# B&R Automation Studio project EFI
Automation Studio 4.12.6.106; Program for EFI Printing Machines; technology packages: Acp10Arnc0 5.21.2, mapp 5.21.0, mappView 5.21.0

## Configuration 1BK2Bar

CPU X20CP1382, AutomationRuntime B4.83, Build 4.1.2, Safety 1.10

### Task classes (Cpu.sw)
```
Cyclic#1 (cycle 4000 us, tolerance 0 us):
  InitSteprs <- ExtPack._Motion.StepperCtrl.StepperCtrl_v1.InitStepperX2XCtrl.prg (BuildOptions=-D _IGNORE_CHECKLIB)
  Stepper3L1 <- ExtPack._Motion.StepperCtrl.StepperCtrl_v1.StepperX2XCtrl.prg (BuildOptions=-D _IGNORE_CHECKLIB)
  Stepper3L2 <- ExtPack._Motion.StepperCtrl.StepperCtrl_v1.StepperX2XCtrl.prg (BuildOptions=-D _IGNORE_CHECKLIB)
  Analog <- (binary) (BuildOptions=-D _IGNORE_CHECKLIB)
  Visu_Inks <- (binary) (BuildOptions=-D _IGNORE_CHECKLIB)
  Slave_mbus <- (binary) (BuildOptions=-D _IGNORE_CHECKLIB)
Cyclic#2 (cycle 12000 us, tolerance 0 us):
  Initialize <- Printer.Config.Initialize.prg (BuildOptions=-D _IGNORE_CHECKLIB)
  InitAxis <- ExtPack._Motion.AxisCtrl.AxisCtrl_v2.InitAxisControl.prg (BuildOptions=-D _IGNORE_CHECKLIB)
  Belt <- ExtPack._Motion.AxisCtrl.AxisCtrl_v2.AxisCtrl.prg (BuildOptions=-D _IGNORE_CHECKLIB)
  BK_A <- ExtPack._Motion.AxisCtrl.AxisCtrl_v2.AxisCtrl.prg (BuildOptions=-D _IGNORE_CHECKLIB)
  Stepper3L <- ExtPack._Motion.AxisCtrl.AxisCtrl_v2.AxisCtrl.prg (BuildOptions=-D _IGNORE_CHECKLIB)
  Gear3L <- ExtPack._Motion.AxisCtrl.AxisCtrl_v2.AxisCtrl.prg (BuildOptions=-D _IGNORE_CHECKLIB)
  InitIcla <- ExtPack._Motion.IclaCtrl.IclaCtrl_v4.InitIclaCtrl.prg (BuildOptions=-D _IGNORE_CHECKLIB)
  IclaBK_A <- ExtPack._Motion.IclaCtrl.IclaCtrl_v4.IclaCtrl.prg (BuildOptions=-D _IGNORE_CHECKLIB)
  Analog_Fas <- ExtPack._Media.AnalogThicknessCtrl.AnalogThicknessCtrl_v1.Analog_Fast.prg (BuildOptions=-D _IGNORE_CHECKLIB)
  nSens_Fast <- ExtPack._Media.nSensorCtrl.nSensorCtrl_v2.nSensorCtrl_Fast.prg (BuildOptions=-D _IGNORE_CHECKLIB)
  Thick_Fast <- ExtPack._Media.ThicknessCtrl.ThicknessCtrl_v2.ThicknessCtrl_Fast.prg (BuildOptions=-D _IGNORE_CHECKLIB)
Cyclic#4 (cycle 32000 us, tolerance 32000 us):
  PhysInput <- Printer.PhysicalMapping.PhysicalMapInputs.prg (BuildOptions=-D _IGNORE_CHECKLIB)
  BlockInp <- Printer.BlockSignalsManager.BlockInputsMapping.prg (BuildOptions=-D _IGNORE_CHECKLIB)  // Physical inputs/outputs block
  ThickPos <- ExtPack._Media.ThicknessCtrl.ThicknessCtrl_v2.ThicknessCtrl.prg (BuildOptions=-D _IGNORE_CHECKLIB)  // Thickness array manager
  Mach_Fast <- Printer.MachineCtrl.MachineCtrl_Fast.prg (BuildOptions=-D _IGNORE_CHECKLIB)
  BeltCtrl <- ExtPack._Transport.BeltCtrl.BeltCtrl_v1.BeltCtrl.prg (BuildOptions=-D _IGNORE_CHECKLIB)  // Belt program
  InitBlockC <- ExtPack.BlockCtrl.BlockCtrl_v1.InitBlockCtrl.prg (BuildOptions=-D _IGNORE_CHECKLIB)  // Init blocks
  Block_BK1 <- ExtPack.BlockCtrl.BlockCtrl_v1.BlockCtrl.prg (BuildOptions=-D _IGNORE_CHECKLIB)
  AnalogThic <- ExtPack._Media.AnalogThicknessCtrl.AnalogThicknessCtrl_v1.AnalogThickness.prg (BuildOptions=-D _IGNORE_CHECKLIB)
  nSensorCtr <- ExtPack._Media.nSensorCtrl.nSensorCtrl_v2.nSensorCtrl.prg (BuildOptions=-D _IGNORE_CHECKLIB)
  InitChille <- ExtPack._Extras.ChillerCtrl.ChillerCtrl_v2.InitChiller.prg (BuildOptions=-D _IGNORE_CHECKLIB)
  ChillCtr1 <- ExtPack._Extras.ChillerCtrl.ChillerCtrl_v2.ChillerCtrl.prg (BuildOptions=-D _IGNORE_CHECKLIB)
  BlockOut <- Printer.BlockSignalsManager.BlockOutputsMapping.prg (BuildOptions=-D _IGNORE_CHECKLIB)  // Physical HW outputs
  PhysOutput <- Printer.PhysicalMapping.PhysicalMapOutputs.prg (BuildOptions=-D _IGNORE_CHECKLIB)
Cyclic#5 (cycle 80000 us, tolerance 80000 us):
  InksInputs <- Printer.InksSignals.InksInputs.prg (BuildOptions=-D _IGNORE_CHECKLIB)  // Physical inputs inks
  InitIndex <- ExtPack.InksCtrl.InksCtrl_v3.InitInksCtrl.prg (BuildOptions=-D _IGNORE_CHECKLIB)
  Inks_01 <- ExtPack.InksCtrl.InksCtrl_v3.InksCtrl.prg (BuildOptions=-D _IGNORE_CHECKLIB)
  Inks_02 <- ExtPack.InksCtrl.InksCtrl_v3.InksCtrl.prg (BuildOptions=-D _IGNORE_CHECKLIB)
  InksOutput <- Printer.InksSignals.InksOutputs.prg (BuildOptions=-D _IGNORE_CHECKLIB)  // Physical outputs inks
  SafetySamp <- AsSafetySolution.SafetySample.prg (BuildOptions=-D _IGNORE_CHECKLIB)
  EventLogGe <- ExtPack._Tools.EventLog.EventLog_v1.EventLogGen.prg (BuildOptions=-D _IGNORE_CHECKLIB)
  SavePerman <- Printer.Config.SavePermanent.prg (BuildOptions=-D _IGNORE_CHECKLIB)
Cyclic#6 (cycle 88000 us, tolerance 88000 us):
  Mach_Conf <- Printer.Config.MachineConfigurator.prg (BuildOptions=-D _IGNORE_CHECKLIB)  // Printer configurator program
  Mach_Slow <- Printer.MachineCtrl.MachineCtrl_Slow.prg (BuildOptions=-D _IGNORE_CHECKLIB)
Cyclic#7 (cycle 44000 us, tolerance 88000 us):
  PLC2Kernel <- Printer.Comms.PLC2Kernel.prg (BuildOptions=-D _IGNORE_CHECKLIB)  // Comn PLC to kernel
  ServModbus <- ExtPack._Comms.ModbusComms.ModbusComms_v1.ServModbus.prg (BuildOptions=-D _IGNORE_CHECKLIB)
  Kernel2PLC <- Printer.Comms.Kernel2PLC.prg (BuildOptions=-D _IGNORE_CHECKLIB)  // Comns Kernel to PLC
Cyclic#8 (cycle 200000 us):
  NwSNTPClie <- ExtPack._Comms.SNTPClient.SNTPClient_v1.NwSNTPClient.prg [disabled] (BuildOptions=-D _IGNORE_CHECKLIB)
DataObjects: Acp10sys, assl1
NcDataObjects: AcpErrTxt <- AxisTables.AcpErrTxt.dob, acp10etxen <- AxisTables.acp10etxen.dob, BeltP4_a <- AxisTables.BeltP4_a.dob, BeltP4_i <- AxisTables.BeltP4_i.dob, BeltShield <- AxisTables.BeltShield_a.dob, BeltShiel1 <- AxisTables.BeltShield_i.dob, BK1_a <- AxisTables.BK1_a.dob, BK1_i <- AxisTables.BK1_i.dob, SM_a <- AxisTables.SM_a.dob, SM_i <- AxisTables.SM_i.dob
Binaries: udbdef, TCData, mvLoader, TCLang, Acp10map, acp10cfg, iomap, User, ashwac, arconfig, Role, ashwd, sysconf, asfw, vccnum, vcpdvnc, Visu02, vccalarm, vccovl, vcshared, vcfile, Panel101, vccstr, vccline, arial, vcpfx20, vcchtml, vcgclass, vccbtn, vcrt, Visu03, vcctext, vcclbox, Panel102, vccbmp, vcfntttf, vcctrend, vcalarm, vcdsint, vcnet, vccshape, arialbd, vctcal, Panel103, vcmgr, vcdsloc, Visu01, vcpkat, vccurl, vccdt, vccbar, vcpdsw, vcxml, vcbclass, Diagn01, vccslider, vccddbox, Diagn02, vccpopup, vcchspot, Diagn03
Libraries: AsCANopen, FBs, Functions, ConvertFun, runtime, brsystem, sys_lib, standard, AsSafety, FileIO, AsXml, astime, asstring, AsFifo, NcGlobal, AsBrStr, MTBasics, MTTypes, MTFilter, AsTCP, AsIecCon, AsIOAcc, AsBrMath, AsEPL, ArEventLog, Acp10_MC, Acp10man, Acp10par, Acp10sim, Acp10sdc, DataObj, EvLogLib, BRSE_MB, BRSE_MBT, AxisFunc, AsSem, AsARCfg, ThickLib, powerlnk, arproject, arssl, asopcuas, asopcuac, vcresman, ashw
```

### Hardware
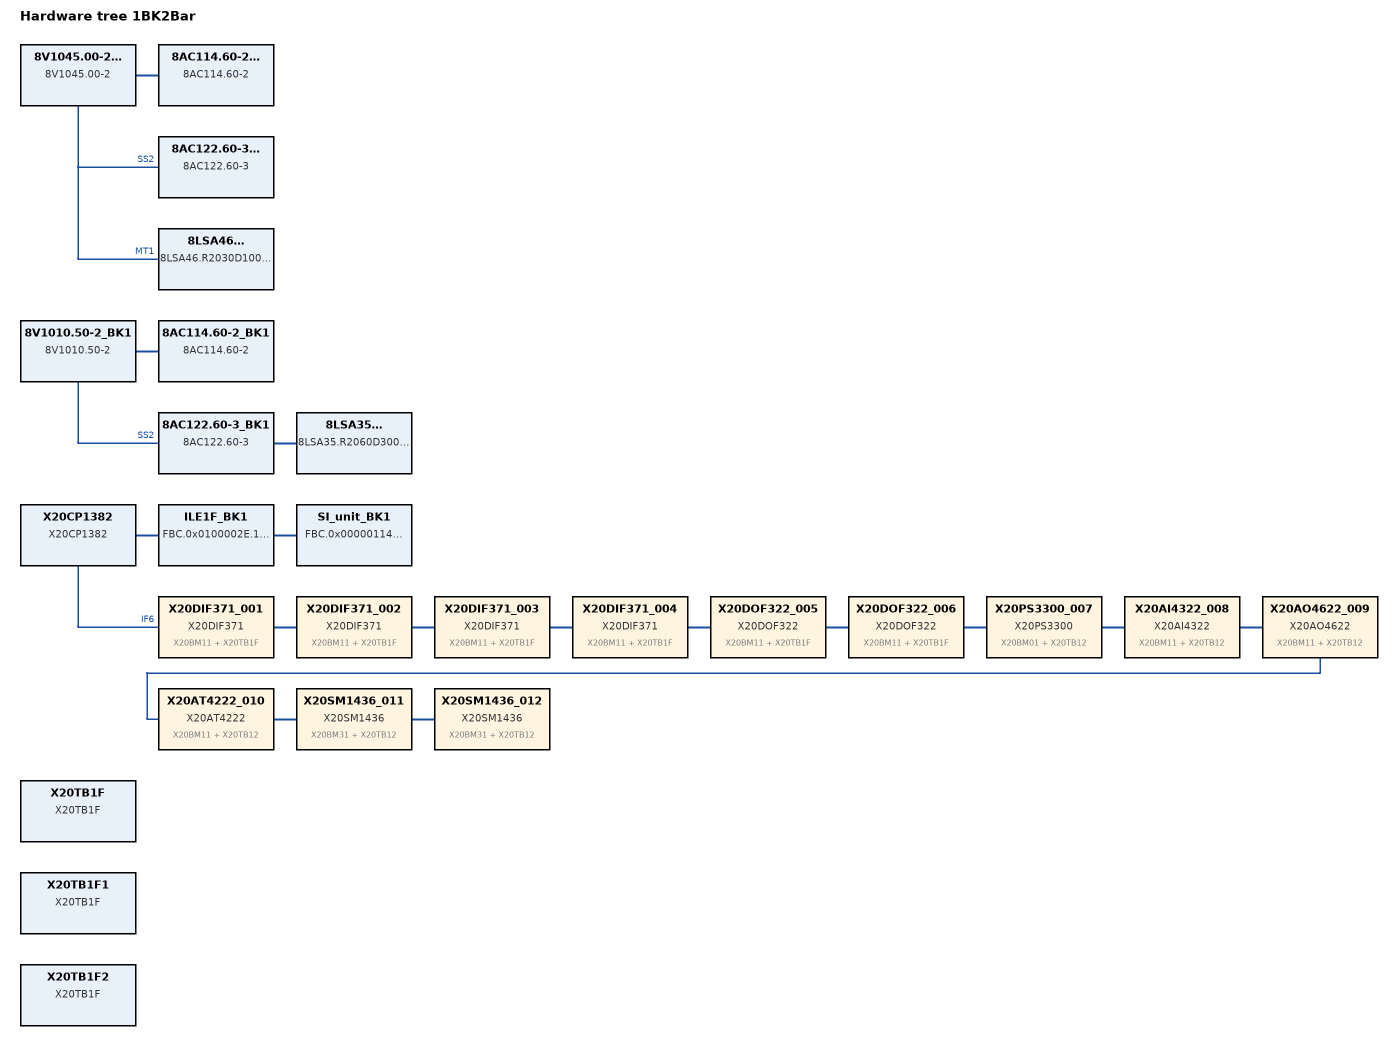
```
8AC114.60-2_BELT : 8AC114.60-2 v1.0.0.8  [SS -> 8V1045.00-2_BELT.SS1; PLK1 -> 8AC114.60-2_BK1.PLK2 (NodeNumber=1) [Cable Type=PowerlinkCable, Length=10, Version=1.0.0.3]]
8AC114.60-2_BK1 : 8AC114.60-2 v1.0.0.8  [SS -> 8V1010.50-2_BK1.SS1; PLK1 -> X20CP1382.IF3 (NodeNumber=2) [Cable Type=PowerlinkCable, Length=10, Version=1.0.0.3]; PLK2 -> 8AC114.60-2_BELT.PLK1 (NodeNumber=2) [Cable Type=PowerlinkCable, Length=10, Version=1.0.0.3]]
8AC122.60-3_BELT : 8AC122.60-3 v2.2.0.0  [SS -> 8V1045.00-2_BELT.SS2]
8AC122.60-3_BK1 : 8AC122.60-3 v2.2.0.0  [SS -> 8V1010.50-2_BK1.SS2]
8LSA35.R2060D300-3 : 8LSA35.R2060D300-3 v1.0.4.39  [EC -> 8AC122.60-3_BK1.EC; MT -> 8V1010.50-2_BK1.MT1]
8LSA46.R2030D100-3 : 8LSA46.R2030D100-3 v2.2.0.0  [MT -> 8V1045.00-2_BELT.MT1]
8V1010.50-2_BK1 : 8V1010.50-2 v2.2.0.0
  SinglePhaseOperation = on
  BothEndSwitchesAreNormallyOpen_r1 = on
  QuickStopIsNormallyOpen_r1 = on
8V1045.00-2_BELT : 8V1045.00-2 v2.2.0.0
ILE1F_BK1 : FBC.0x0100002E.1.SEILE1F_0110E v1.10 (OrderNumber=ILE1F)  [CAN1 -> X20CP1382.IF7 (NodeNumber=5)]
  p1403_transmissionselection = 1
  plifeguarding_guardtime = 500
  plifeguarding_retryfactor = 10
  p3001_parametername = mandatory
  p3001_objecttype = 9
  p3001_subnumber = 0x3
  p3001_parametervalue = 
  p3001_objflags = 0
  p3001sub0_parametername = number of entries
  p3001sub0_objecttype = 7
  p3001sub0_datatype = 5
  p3001sub0_accesstype = ro
  p3001sub0_pdomapping = 0
  p3001sub1_parametername = Config.PrgNo
  p3001sub1_objecttype = 7
  p3001sub1_datatype = 7
  p3001sub1_lowlimit = 
  p3001sub1_highlimit = 
  p3001sub1_accesstype = ro
  p3001sub1_pdomapping = 0
  p3001sub2_parametername = Config.PrgVer
  p3001sub2_objecttype = 7
  p3001sub2_datatype = 7
  p3001sub2_lowlimit = 
  p3001sub2_highlimit = 
  p3001sub2_accesstype = ro
  p3001sub2_pdomapping = 0
  p300b_parametername = system settings
  p300b_objecttype = 9
  p300b_subnumber = 0x7
  p300b_parametervalue = 
  p300b_objflags = 0
  p300bsub0_parametername = number of entries
  p300bsub0_objecttype = 7
  p300bsub0_datatype = 5
  p300bsub0_accesstype = ro
  p300bsub0_pdomapping = 0
  p300bsub1_parametername = Settings.name1
  p300bsub1_objecttype = 7
  p300bsub1_datatype = 7
  p300bsub1_lowlimit = 
  p300bsub1_highlimit = 
  p300bsub1_accesstype = rw
  p300bsub1_pdomapping = 0
  p300bsub1_parametervalue = 
  p300bsub1_objflags = 0
  p300bsub2_parametername = Settings.name2
  p300bsub2_objecttype = 7
  p300bsub2_datatype = 7
  p300bsub2_lowlimit = 
  p300bsub2_highlimit = 
  p300bsub2_accesstype = rw
  p300bsub2_pdomapping = 0
  p300bsub2_parametervalue = 
  p300bsub2_objflags = 0
  p300bsub6_parametername = Commands.eeprSave
  p300bsub6_objecttype = 7
  p300bsub6_datatype = 6
  p300bsub6_lowlimit = 
  p300bsub6_highlimit = 
  p300bsub6_accesstype = rw
  p300bsub6_pdomapping = 0
  p300bsub6_parametervalue = 1
  p300bsub6_objflags = 0
  p300bsub7_parametername = Commands.stateSave
  p300bsub7_objecttype = 7
  p300bsub7_datatype = 6
  p300bsub7_lowlimit = 
  p300bsub7_highlimit = 
  p300bsub7_accesstype = ro
  p300bsub7_pdomapping = 0
  p300bsub8_parametername = Commands.default
  p300bsub8_objecttype = 7
  p300bsub8_datatype = 6
  p300bsub8_lowlimit = 
  p300bsub8_highlimit = 
  p300bsub8_accesstype = rw
  p300bsub8_pdomapping = 0
  p300bsub8_parametervalue = 
  p300bsub8_objflags = 0
  p300bsub9_parametername = Commands.stateDef
  p300bsub9_objecttype = 7
  p300bsub9_datatype = 6
  p300bsub9_lowlimit = 
  p300bsub9_highlimit = 
  p300bsub9_accesstype = ro
  p300bsub9_pdomapping = 0
  p300f_parametername = controller  settings
  p300f_objecttype = 9
  p300f_subnumber = 0xE
  p300f_parametervalue = 
  p300f_objflags = 0
  p300fsub0_parametername = number of entries
  p300fsub0_objecttype = 7
  p300fsub0_datatype = 5
  p300fsub0_accesstype = ro
  p300fsub0_pdomapping = 0
  p300fsub1_parametername = Config.I_nomDrv
  p300fsub1_objecttype = 7
  p300fsub1_datatype = 6
  p300fsub1_accesstype = ro
  p300fsub1_pdomapping = 0
  p300fsub2_parametername = Config.I_maxDrv
  p300fsub2_objecttype = 7
  p300fsub2_datatype = 6
  p300fsub2_accesstype = ro
  p300fsub2_pdomapping = 0
  p300fsub3_parametername = Settings.I_max
  p300fsub3_objecttype = 7
  p300fsub3_datatype = 6
  p300fsub3_accesstype = rw
  p300fsub3_pdomapping = 0
  p300fsub3_parametervalue = 60
  p300fsub3_objflags = 0
  p300fsub5_parametername = Settings.I_maxBlk
  p300fsub5_objecttype = 7
  p300fsub5_datatype = 6
  p300fsub5_lowlimit = 
  p300fsub5_highlimit = 
  p300fsub5_accesstype = rw
  p300fsub5_pdomapping = 0
  p300fsub5_parametervalue = 20
  p300fsub5_objflags = 0
  p300fsub7_parametername = Settings.p_maxDiff
  p300fsub7_objecttype = 7
  p300fsub7_datatype = 6
  p300fsub7_lowlimit = 
  p300fsub7_highlimit = 
  p300fsub7_accesstype = rw
  p300fsub7_pdomapping = 0
  p300fsub7_parametervalue = 24
  p300fsub7_objflags = 0
  p300fsub8_parametername = Control.KPn
  p300fsub8_objecttype = 7
  p300fsub8_datatype = 6
  p300fsub8_lowlimit = 
  p300fsub8_highlimit = 
  p300fsub8_accesstype = rw
  p300fsub8_pdomapping = 0
  p300fsub8_parametervalue = 60
  p300fsub8_objflags = 0
  p300fsub9_parametername = Control.TNn
  p300fsub9_objecttype = 7
  p300fsub9_datatype = 6
  p300fsub9_lowlimit = 
  p300fsub9_highlimit = 
  p300fsub9_accesstype = rw
  p300fsub9_pdomapping = 0
  p300fsub9_parametervalue = 10000
  p300fsub9_objflags = 0
  p300fsuba_parametername = Control.KPp
  p300fsuba_objecttype = 7
  p300fsuba_datatype = 6
  p300fsuba_lowlimit = 
  p300fsuba_highlimit = 
  p300fsuba_accesstype = rw
  p300fsuba_pdomapping = 0
  p300fsuba_parametervalue = 300
  p300fsuba_objflags = 0
  p300fsubb_parametername = Control.KFPp
  p300fsubb_objecttype = 7
  p300fsubb_datatype = 6
  p300fsubb_lowlimit = 
  p300fsubb_highlimit = 
  p300fsubb_accesstype = rw
  p300fsubb_pdomapping = 0
  p300fsubb_parametervalue = 32767
  p300fsubb_objflags = 0
  p300fsubc_parametername = Settings.T_block
  p300fsubc_objecttype = 7
  p300fsubc_datatype = 6
  p300fsubc_lowlimit = 
  p300fsubc_highlimit = 
  p300fsubc_accesstype = rw
  p300fsubc_pdomapping = 0
  p300fsubc_parametervalue = 100
  p300fsubc_objflags = 0
  p300fsubd_parametername = Status.p_difPeak
  p300fsubd_objecttype = 7
  p300fsubd_datatype = 7
  p300fsubd_lowlimit = 
  p300fsubd_highlimit = 
  p300fsubd_accesstype = rw
  p300fsubd_pdomapping = 0
  p300fsubd_parametervalue = 
  p300fsubd_objflags = 0
  p300fsubf_parametername = Settings.p_win
  p300fsubf_objecttype = 7
  p300fsubf_datatype = 6
  p300fsubf_lowlimit = 
  p300fsubf_highlimit = 
  p300fsubf_accesstype = rw
  p300fsubf_pdomapping = 0
  p300fsubf_parametervalue = 1
  p300fsubf_objflags = 0
  p300fsub10_parametername = Settings.p_winTime
  p300fsub10_objecttype = 7
  p300fsub10_datatype = 6
  p300fsub10_lowlimit = 
  p300fsub10_highlimit = 
  p300fsub10_accesstype = rw
  p300fsub10_pdomapping = 0
  p300fsub10_parametervalue = 0
  p300fsub10_objflags = 0
  p3016_parametername = rs485
  p3016_objecttype = 9
  p3016_subnumber = 0x4
  p3016_parametervalue = 
  p3016_objflags = 0
  p3016sub0_parametername = number of entries
  p3016sub0_objecttype = 7
  p3016sub0_datatype = 5
  p3016sub0_accesstype = ro
  p3016sub0_pdomapping = 0
  p3016sub1_parametername = RS485.serBaud
  p3016sub1_objecttype = 7
  p3016sub1_datatype = 6
  p3016sub1_lowlimit = 
  p3016sub1_highlimit = 
  p3016sub1_accesstype = rw
  p3016sub1_pdomapping = 0
  p3016sub1_parametervalue = 
  p3016sub1_objflags = 0
  p3016sub2_parametername = RS485.serAdr
  p3016sub2_objecttype = 7
  p3016sub2_datatype = 6
  p3016sub2_lowlimit = 
  p3016sub2_highlimit = 
  p3016sub2_accesstype = rw
  p3016sub2_pdomapping = 0
  p3016sub2_parametervalue = 
  p3016sub2_objflags = 0
  p3016sub3_parametername = RS485.serFormat
  p3016sub3_objecttype = 7
  p3016sub3_datatype = 6
  p3016sub3_lowlimit = 
  p3016sub3_highlimit = 
  p3016sub3_accesstype = rw
  p3016sub3_pdomapping = 0
  p3016sub3_parametervalue = 
  p3016sub3_objflags = 0
  p3017_parametername = can
  p3017_objecttype = 9
  p3017_subnumber = 0x3
  p3017_parametervalue = 
  p3017_objflags = 0
  p3017sub0_parametername = number of entries
  p3017sub0_objecttype = 7
  p3017sub0_datatype = 5
  p3017sub0_accesstype = ro
  p3017sub0_pdomapping = 0
  p3017sub2_parametername = CAN.canAddr
  p3017sub2_objecttype = 7
  p3017sub2_datatype = 6
  p3017sub2_lowlimit = 
  p3017sub2_highlimit = 
  p3017sub2_accesstype = rw
  p3017sub2_pdomapping = 0
  p3017sub2_parametervalue = 
  p3017sub2_objflags = 0
  p3017sub3_parametername = CAN.canBaud
  p3017sub3_objecttype = 7
  p3017sub3_datatype = 6
  p3017sub3_lowlimit = 
  p3017sub3_highlimit = 
  p3017sub3_accesstype = rw
  p3017sub3_pdomapping = 0
  p3017sub3_parametervalue = 
  p3017sub3_objflags = 0
  p301c_parametername = settings1
  p301c_objecttype = 9
  p301c_subnumber = 0xF
  p301c_parametervalue = 
  p301c_objflags = 0
  p301csub0_parametername = number of entries
  p301csub0_objecttype = 7
  p301csub0_datatype = 5
  p301csub0_accesstype = ro
  p301csub0_pdomapping = 0
  p301csub3_parametername = Status.xMode_act
  p301csub3_objecttype = 7
  p301csub3_datatype = 6
  p301csub3_lowlimit = 
  p301csub3_highlimit = 
  p301csub3_accesstype = ro
  p301csub3_pdomapping = 0
  p301csub6_parametername = Motion.invertDir
  p301csub6_objecttype = 7
  p301csub6_datatype = 6
  p301csub6_lowlimit = 
  p301csub6_highlimit = 
  p301csub6_accesstype = rw
  p301csub6_pdomapping = 0
  p301csub6_parametervalue = 0
  p301csub6_objflags = 0
  p301csuba_parametername = Status.WarnSig
  p301csuba_objecttype = 7
  p301csuba_datatype = 6
  p301csuba_lowlimit = 
  p301csuba_highlimit = 
  p301csuba_accesstype = ro
  p301csuba_pdomapping = 0
  p301csubb_parametername = Settings.WarnOvrun
  p301csubb_objecttype = 7
  p301csubb_datatype = 6
  p301csubb_lowlimit = 
  p301csubb_highlimit = 
  p301csubb_accesstype = rw
  p301csubb_pdomapping = 0
  p301csubb_parametervalue = 0
  p301csubb_objflags = 0
  p301csubd_parametername = Settings.SignEnabl
  p301csubd_objecttype = 7
  p301csubd_datatype = 6
  p301csubd_lowlimit = 
  p301csubd_highlimit = 
  p301csubd_accesstype = rw
  p301csubd_pdomapping = 0
  p301csubd_parametervalue = 3
  p301csubd_objflags = 0
  p301csube_parametername = Settings.SignLevel
  p301csube_objecttype = 7
  p301csube_datatype = 6
  p301csube_lowlimit = 
  p301csube_highlimit = 
  p301csube_accesstype = rw
  p301csube_pdomapping = 0
  p301csube_parametervalue = 0
  p301csube_objflags = 0
  p301csubf_parametername = Status.Sign_SR
  p301csubf_objecttype = 7
  p301csubf_datatype = 6
  p301csubf_lowlimit = 
  p301csubf_highlimit = 
  p301csubf_accesstype = ro
  p301csubf_pdomapping = 0
  p301csub11_parametername = Status.FltSig
  p301csub11_objecttype = 7
  p301csub11_datatype = 7
  p301csub11_lowlimit = 
  p301csub11_highlimit = 
  p301csub11_accesstype = ro
  p301csub11_pdomapping = 0
  p301csub12_parametername = Status.FltSig_SR
  p301csub12_objecttype = 7
  p301csub12_datatype = 7
  p301csub12_lowlimit = 
  p301csub12_highlimit = 
  p301csub12_accesstype = ro
  p301csub12_pdomapping = 0
  p301csub13_parametername = Status.action_st
  p301csub13_objecttype = 7
  p301csub13_datatype = 6
  p301csub13_lowlimit = 
  p301csub13_highlimit = 
  p301csub13_accesstype = ro
  p301csub13_pdomapping = 0
  p301csub15_parametername = Motion.dec_Stop
  p301csub15_objecttype = 7
  p301csub15_datatype = 7
  p301csub15_lowlimit = 
  p301csub15_highlimit = 
  p301csub15_accesstype = rw
  p301csub15_pdomapping = 0
  p301csub15_parametervalue = 4960
  p301csub15_objflags = 0
  p301csub18_parametername = Settings.Flt_pDiff
  p301csub18_objecttype = 7
  p301csub18_datatype = 6
  p301csub18_lowlimit = 
  p301csub18_highlimit = 
  p301csub18_accesstype = rw
  p301csub18_pdomapping = 0
  p301csub18_parametervalue = 3
  p301csub18_objflags = 0
  p301d_parametername = settings2
  p301d_objecttype = 9
  p301d_subnumber = 0x4
  p301d_parametervalue = 
  p301d_objflags = 0
  p301dsub0_parametername = number of entries
  p301dsub0_objecttype = 7
  p301dsub0_datatype = 5
  p301dsub0_accesstype = ro
  p301dsub0_pdomapping = 0
  p301dsub2_parametername = Config.ResolutM
  p301dsub2_objecttype = 7
  p301dsub2_datatype = 6
  p301dsub2_accesstype = ro
  p301dsub2_pdomapping = 0
  p301dsub17_parametername = Motion.v_target0
  p301dsub17_objecttype = 7
  p301dsub17_datatype = 6
  p301dsub17_accesstype = rw
  p301dsub17_pdomapping = 0
  p301dsub17_parametervalue = 1000
  p301dsub17_objflags = 0
  p301dsub1a_parametername = Motion.acc
  p301dsub1a_objecttype = 7
  p301dsub1a_datatype = 7
  p301dsub1a_lowlimit = 
  p301dsub1a_highlimit = 
  p301dsub1a_accesstype = rw
  p301dsub1a_pdomapping = 0
  p301dsub1a_parametervalue = 2442
  p301dsub1a_objflags = 0
  p301e_parametername = pdo data
  p301e_objecttype = 9
  p301e_subnumber = 0xC
  p301e_parametervalue = 
  p301e_objflags = 0
  p301esub0_parametername = number of entries
  p301esub0_objecttype = 7
  p301esub0_datatype = 5
  p301esub0_accesstype = ro
  p301esub0_pdomapping = 0
  p301esubb_parametername = Status.ModeError
  p301esubb_objecttype = 7
  p301esubb_datatype = 6
  p301esubb_lowlimit = 
  p301esubb_highlimit = 
  p301esubb_accesstype = ro
  p301esubb_pdomapping = 0
  p301f_parametername = status
  p301f_objecttype = 9
  p301f_subnumber = 0x11
  p301f_parametervalue = 
  p301f_objflags = 0
  p301fsub0_parametername = number of entries
  p301fsub0_objecttype = 7
  p301fsub0_datatype = 5
  p301fsub0_accesstype = ro
  p301fsub0_pdomapping = 0
  p301fsub1_parametername = Status.v_ref
  p301fsub1_objecttype = 7
  p301fsub1_datatype = 4
  p301fsub1_lowlimit = 
  p301fsub1_highlimit = 
  p301fsub1_accesstype = ro
  p301fsub1_pdomapping = 0
  p301fsub2_parametername = Status.v_act
  p301fsub2_objecttype = 7
  p301fsub2_datatype = 4
  p301fsub2_lowlimit = 
  p301fsub2_highlimit = 
  p301fsub2_accesstype = ro
  p301fsub2_pdomapping = 0
  p301fsub5_parametername = Status.p_ref
  p301fsub5_objecttype = 7
  p301fsub5_datatype = 4
  p301fsub5_lowlimit = 
  p301fsub5_highlimit = 
  p301fsub5_accesstype = ro
  p301fsub5_pdomapping = 0
  p301fsub6_parametername = Status.p_act
  p301fsub6_objecttype = 7
  p301fsub6_datatype = 4
  p301fsub6_lowlimit = 
  p301fsub6_highlimit = 
  p301fsub6_accesstype = ro
  p301fsub6_pdomapping = 0
  p301fsub7_parametername = Status.p_dif
  p301fsub7_objecttype = 7
  p301fsub7_datatype = 4
  p301fsub7_lowlimit = 
  p301fsub7_highlimit = 
  p301fsub7_accesstype = ro
  p301fsub7_pdomapping = 0
  p301fsub8_parametername = Status.n_ref
  p301fsub8_objecttype = 7
  p301fsub8_datatype = 3
  p301fsub8_lowlimit = 
  p301fsub8_highlimit = 
  p301fsub8_accesstype = ro
  p301fsub8_pdomapping = 0
  p301fsub9_parametername = Status.n_act
  p301fsub9_objecttype = 7
  p301fsub9_datatype = 3
  p301fsub9_lowlimit = 
  p301fsub9_highlimit = 
  p301fsub9_accesstype = ro
  p301fsub9_pdomapping = 0
  p301fsubc_parametername = Status.I_act
  p301fsubc_objecttype = 7
  p301fsubc_datatype = 3
  p301fsubc_lowlimit = 
  p301fsubc_highlimit = 
  p301fsubc_accesstype = ro
  p301fsubc_pdomapping = 0
  p301fsub14_parametername = Status.UDC_act
  p301fsub14_objecttype = 7
  p301fsub14_datatype = 6
  p301fsub14_lowlimit = 
  p301fsub14_highlimit = 
  p301fsub14_accesstype = ro
  p301fsub14_pdomapping = 0
  p301fsub19_parametername = Status.TPA_act
  p301fsub19_objecttype = 7
  p301fsub19_datatype = 6
  p301fsub19_lowlimit = 
  p301fsub19_highlimit = 
  p301fsub19_accesstype = ro
  p301fsub19_pdomapping = 0
  p301fsub1c_parametername = Status.v_pref
  p301fsub1c_objecttype = 7
  p301fsub1c_datatype = 4
  p301fsub1c_lowlimit = 
  p301fsub1c_highlimit = 
  p301fsub1c_accesstype = ro
  p301fsub1c_pdomapping = 0
  p301fsub1e_parametername = Status.p_target
  p301fsub1e_objecttype = 7
  p301fsub1e_datatype = 4
  p301fsub1e_lowlimit = 
  p301fsub1e_highlimit = 
  p301fsub1e_accesstype = ro
  p301fsub1e_pdomapping = 0
  p301fsub1f_parametername = Status.p_profile
  p301fsub1f_objecttype = 7
  p301fsub1f_datatype = 4
  p301fsub1f_lowlimit = 
  p301fsub1f_highlimit = 
  p301fsub1f_accesstype = ro
  p301fsub1f_pdomapping = 0
  p301fsub23_parametername = Status.n_profile
  p301fsub23_objecttype = 7
  p301fsub23_datatype = 3
  p301fsub23_lowlimit = 
  p301fsub23_highlimit = 
  p301fsub23_accesstype = ro
  p301fsub23_pdomapping = 0
  p301fsub26_parametername = Status.n_target
  p301fsub26_objecttype = 7
  p301fsub26_datatype = 3
  p301fsub26_lowlimit = 
  p301fsub26_highlimit = 
  p301fsub26_accesstype = ro
  p301fsub26_pdomapping = 0
  p301fsub2d_parametername = Status.n_pref
  p301fsub2d_objecttype = 7
  p301fsub2d_datatype = 3
  p301fsub2d_lowlimit = 
  p301fsub2d_highlimit = 
  p301fsub2d_accesstype = ro
  p301fsub2d_pdomapping = 0
  p3020_parametername = error
  p3020_objecttype = 9
  p3020_subnumber = 0x5
  p3020_parametervalue = 
  p3020_objflags = 0
  p3020sub0_parametername = number of entries
  p3020sub0_objecttype = 7
  p3020sub0_datatype = 5
  p3020sub0_accesstype = ro
  p3020sub0_pdomapping = 0
  p3020sub1_parametername = ErrorMemAvailable
  p3020sub1_objecttype = 7
  p3020sub1_datatype = 6
  p3020sub1_lowlimit = 
  p3020sub1_highlimit = 
  p3020sub1_accesstype = ro
  p3020sub1_pdomapping = 0
  p3020sub2_parametername = Commands.del_err
  p3020sub2_objecttype = 7
  p3020sub2_datatype = 6
  p3020sub2_lowlimit = 
  p3020sub2_highlimit = 
  p3020sub2_accesstype = rw
  p3020sub2_pdomapping = 0
  p3020sub2_parametervalue = 
  p3020sub2_objflags = 0
  p3020sub6_parametername = PowerOnCount
  p3020sub6_objecttype = 7
  p3020sub6_datatype = 7
  p3020sub6_lowlimit = 
  p3020sub6_highlimit = 
  p3020sub6_accesstype = ro
  p3020sub6_pdomapping = 0
  p3020sub7_parametername = Status.StopFault
  p3020sub7_objecttype = 7
  p3020sub7_datatype = 6
  p3020sub7_lowlimit = 
  p3020sub7_highlimit = 
  p3020sub7_accesstype = ro
  p3020sub7_pdomapping = 0
  p3021_parametername = io
  p3021_objecttype = 9
  p3021_subnumber = 0x4
  p3021_parametervalue = 
  p3021_objflags = 0
  p3021sub0_parametername = number of entries
  p3021sub0_objecttype = 7
  p3021sub0_datatype = 5
  p3021sub0_accesstype = ro
  p3021sub0_pdomapping = 0
  p3021sub1_parametername = I/O.IO_act
  p3021sub1_objecttype = 7
  p3021sub1_datatype = 6
  p3021sub1_lowlimit = 
  p3021sub1_highlimit = 
  p3021sub1_accesstype = rw
  p3021sub1_pdomapping = 0
  p3021sub1_parametervalue = 
  p3021sub1_objflags = 0
  p3021sub7_parametername = Commands.brake
  p3021sub7_objecttype = 7
  p3021sub7_datatype = 6
  p3021sub7_lowlimit = 
  p3021sub7_highlimit = 
  p3021sub7_accesstype = rw
  p3021sub7_pdomapping = 0
  p3021sub7_parametervalue = 
  p3021sub7_objflags = 0
  p3021sub8_parametername = Status.brake
  p3021sub8_objecttype = 7
  p3021sub8_datatype = 6
  p3021sub8_lowlimit = 
  p3021sub8_highlimit = 
  p3021sub8_accesstype = ro
  p3021sub8_pdomapping = 0
  p3022_parametername = io definitions
  p3022_objecttype = 9
  p3022_subnumber = 0x6
  p3022_parametervalue = 
  p3022_objflags = 0
  p3022sub0_parametername = number of entries
  p3022sub0_objecttype = 7
  p3022sub0_datatype = 5
  p3022sub0_accesstype = ro
  p3022sub0_pdomapping = 0
  p3022sub1_parametername = I/O.IO0_def
  p3022sub1_objecttype = 7
  p3022sub1_datatype = 6
  p3022sub1_lowlimit = 
  p3022sub1_highlimit = 
  p3022sub1_accesstype = rw
  p3022sub1_pdomapping = 0
  p3022sub1_parametervalue = 0
  p3022sub1_objflags = 0
  p3022sub2_parametername = I/O.IO1_def
  p3022sub2_objecttype = 7
  p3022sub2_datatype = 6
  p3022sub2_lowlimit = 
  p3022sub2_highlimit = 
  p3022sub2_accesstype = rw
  p3022sub2_pdomapping = 0
  p3022sub2_parametervalue = 0
  p3022sub2_objflags = 0
  p3022sub3_parametername = I/O.IO2_def
  p3022sub3_objecttype = 7
  p3022sub3_datatype = 6
  p3022sub3_lowlimit = 
  p3022sub3_highlimit = 
  p3022sub3_accesstype = rw
  p3022sub3_pdomapping = 0
  p3022sub3_parametervalue = 0
  p3022sub3_objflags = 0
  p3022sub4_parametername = I/O.IO3_def
  p3022sub4_objecttype = 7
  p3022sub4_datatype = 6
  p3022sub4_lowlimit = 
  p3022sub4_highlimit = 
  p3022sub4_accesstype = rw
  p3022sub4_pdomapping = 0
  p3022sub4_parametervalue = 
  p3022sub4_objflags = 0
  p3022sub7_parametername = I/O.progDelay
  p3022sub7_objecttype = 7
  p3022sub7_datatype = 6
  p3022sub7_lowlimit = 
  p3022sub7_highlimit = 
  p3022sub7_accesstype = rw
  p3022sub7_pdomapping = 0
  p3022sub7_parametervalue = 
  p3022sub7_objflags = 0
  p3023_parametername = ptp
  p3023_objecttype = 9
  p3023_subnumber = 0x6
  p3023_parametervalue = 
  p3023_objflags = 0
  p3023sub0_parametername = number of entries
  p3023sub0_objecttype = 7
  p3023sub0_datatype = 5
  p3023sub0_accesstype = ro
  p3023sub0_pdomapping = 0
  p3023sub1_parametername = PTP.p_absPTP
  p3023sub1_objecttype = 7
  p3023sub1_datatype = 4
  p3023sub1_lowlimit = 
  p3023sub1_highlimit = 
  p3023sub1_accesstype = rw
  p3023sub1_pdomapping = 0
  p3023sub1_parametervalue = 
  p3023sub1_objflags = 0
  p3023sub2_parametername = PTP.StatePTP
  p3023sub2_objecttype = 7
  p3023sub2_datatype = 6
  p3023sub2_lowlimit = 
  p3023sub2_highlimit = 
  p3023sub2_accesstype = ro
  p3023sub2_pdomapping = 0
  p3023sub3_parametername = PTP.p_relPTP
  p3023sub3_objecttype = 7
  p3023sub3_datatype = 4
  p3023sub3_lowlimit = 
  p3023sub3_highlimit = 
  p3023sub3_accesstype = rw
  p3023sub3_pdomapping = 0
  p3023sub3_parametervalue = 
  p3023sub3_objflags = 0
  p3023sub4_parametername = PTP.continue
  p3023sub4_objecttype = 7
  p3023sub4_datatype = 6
  p3023sub4_lowlimit = 
  p3023sub4_highlimit = 
  p3023sub4_accesstype = rw
  p3023sub4_pdomapping = 0
  p3023sub4_parametervalue = 
  p3023sub4_objflags = 0
  p3023sub5_parametername = PTP.v_tarPTP
  p3023sub5_objecttype = 7
  p3023sub5_datatype = 6
  p3023sub5_accesstype = rw
  p3023sub5_pdomapping = 0
  p3023sub5_parametervalue = 
  p3023sub5_objflags = 0
  p3024_parametername = vel
  p3024_objecttype = 9
  p3024_subnumber = 0x3
  p3024_parametervalue = 
  p3024_objflags = 0
  p3024sub0_parametername = number of entries
  p3024sub0_objecttype = 7
  p3024sub0_datatype = 5
  p3024sub0_accesstype = ro
  p3024sub0_pdomapping = 0
  p3024sub1_parametername = VEL.velocity
  p3024sub1_objecttype = 7
  p3024sub1_datatype = 3
  p3024sub1_accesstype = rw
  p3024sub1_pdomapping = 0
  p3024sub1_parametervalue = 
  p3024sub1_objflags = 0
  p3024sub2_parametername = VEL.stateVEL
  p3024sub2_objecttype = 7
  p3024sub2_datatype = 6
  p3024sub2_lowlimit = 
  p3024sub2_highlimit = 
  p3024sub2_accesstype = ro
  p3024sub2_pdomapping = 0
  p3028_parametername = homing
  p3028_objecttype = 9
  p3028_subnumber = 0xB
  p3028_parametervalue = 
  p3028_objflags = 0
  p3028sub0_parametername = number of entries
  p3028sub0_objecttype = 7
  p3028sub0_datatype = 5
  p3028sub0_accesstype = ro
  p3028sub0_pdomapping = 0
  p3028sub1_parametername = Homing.startHome
  p3028sub1_objecttype = 7
  p3028sub1_datatype = 6
  p3028sub1_lowlimit = 
  p3028sub1_highlimit = 
  p3028sub1_accesstype = rw
  p3028sub1_pdomapping = 0
  p3028sub1_parametervalue = 
  p3028sub1_objflags = 0
  p3028sub2_parametername = Homing.stateHome
  p3028sub2_objecttype = 7
  p3028sub2_datatype = 6
  p3028sub2_lowlimit = 
  p3028sub2_highlimit = 
  p3028sub2_accesstype = ro
  p3028sub2_pdomapping = 0
  p3028sub3_parametername = Homing.startSetp
  p3028sub3_objecttype = 7
  p3028sub3_datatype = 4
  p3028sub3_lowlimit = 
  p3028sub3_highlimit = 
  p3028sub3_accesstype = rw
  p3028sub3_pdomapping = 0
  p3028sub3_parametervalue = 
  p3028sub3_objflags = 0
  p3028sub4_parametername = Homing.v_Home
  p3028sub4_objecttype = 7
  p3028sub4_datatype = 6
  p3028sub4_accesstype = rw
  p3028sub4_pdomapping = 0
  p3028sub4_parametervalue = 
  p3028sub4_objflags = 0
  p3028sub5_parametername = Homing.v_outHome
  p3028sub5_objecttype = 7
  p3028sub5_datatype = 6
  p3028sub5_accesstype = rw
  p3028sub5_pdomapping = 0
  p3028sub5_parametervalue = 
  p3028sub5_objflags = 0
  p3028sub6_parametername = Homing.p_outHome
  p3028sub6_objecttype = 7
  p3028sub6_datatype = 4
  p3028sub6_lowlimit = 
  p3028sub6_highlimit = 
  p3028sub6_accesstype = rw
  p3028sub6_pdomapping = 0
  p3028sub6_parametervalue = 
  p3028sub6_objflags = 0
  p3028sub7_parametername = Homing.p_disHome
  p3028sub7_objecttype = 7
  p3028sub7_datatype = 4
  p3028sub7_lowlimit = 
  p3028sub7_highlimit = 
  p3028sub7_accesstype = rw
  p3028sub7_pdomapping = 0
  p3028sub7_parametervalue = 
  p3028sub7_objflags = 0
  p3028sub9_parametername = Homing.RefSwMod
  p3028sub9_objecttype = 7
  p3028sub9_datatype = 6
  p3028sub9_lowlimit = 
  p3028sub9_highlimit = 
  p3028sub9_accesstype = rw
  p3028sub9_pdomapping = 0
  p3028sub9_parametervalue = 
  p3028sub9_objflags = 0
  p3028subb_parametername = Homing.RefAppPos
  p3028subb_objecttype = 7
  p3028subb_datatype = 4
  p3028subb_lowlimit = 
  p3028subb_highlimit = 
  p3028subb_accesstype = rw
  p3028subb_pdomapping = 0
  p3028subb_parametervalue = 
  p3028subb_objflags = 0
  p3028subd_parametername = Homing.refError
  p3028subd_objecttype = 7
  p3028subd_datatype = 6
  p3028subd_lowlimit = 
  p3028subd_highlimit = 
  p3028subd_accesstype = ro
  p3028subd_pdomapping = 0
  p3029_parametername = manual
  p3029_objecttype = 9
  p3029_subnumber = 0x7
  p3029_parametervalue = 
  p3029_objflags = 0
  p3029sub0_parametername = number of entries
  p3029sub0_objecttype = 7
  p3029sub0_datatype = 5
  p3029sub0_accesstype = ro
  p3029sub0_pdomapping = 0
  p3029sub1_parametername = Manual.startMan
  p3029sub1_objecttype = 7
  p3029sub1_datatype = 6
  p3029sub1_lowlimit = 
  p3029sub1_highlimit = 
  p3029sub1_accesstype = rw
  p3029sub1_pdomapping = 0
  p3029sub1_parametervalue = 
  p3029sub1_objflags = 0
  p3029sub2_parametername = Manual.stateMan
  p3029sub2_objecttype = 7
  p3029sub2_datatype = 6
  p3029sub2_lowlimit = 
  p3029sub2_highlimit = 
  p3029sub2_accesstype = ro
  p3029sub2_pdomapping = 0
  p3029sub4_parametername = Manual.n_slowMan
  p3029sub4_objecttype = 7
  p3029sub4_datatype = 6
  p3029sub4_accesstype = rw
  p3029sub4_pdomapping = 0
  p3029sub4_parametervalue = 
  p3029sub4_objflags = 0
  p3029sub5_parametername = Manual.n_fastMan
  p3029sub5_objecttype = 7
  p3029sub5_datatype = 6
  p3029sub5_accesstype = rw
  p3029sub5_pdomapping = 0
  p3029sub5_parametervalue = 
  p3029sub5_objflags = 0
  p3029sub7_parametername = Manual.step_Man
  p3029sub7_objecttype = 7
  p3029sub7_datatype = 6
  p3029sub7_lowlimit = 
  p3029sub7_highlimit = 
  p3029sub7_accesstype = rw
  p3029sub7_pdomapping = 0
  p3029sub7_parametervalue = 
  p3029sub7_objflags = 0
  p3029sub8_parametername = Manual.time_Man
  p3029sub8_objecttype = 7
  p3029sub8_datatype = 6
  p3029sub8_lowlimit = 
  p3029sub8_highlimit = 
  p3029sub8_accesstype = rw
  p3029sub8_pdomapping = 0
  p3029sub8_parametervalue = 
  p3029sub8_objflags = 0
  p3320_parametername = prog io0
  p3320_objecttype = 9
  p3320_subnumber = 0x7
  p3320_parametervalue = 
  p3320_objflags = 0
  p3320sub0_parametername = number of entries
  p3320sub0_objecttype = 7
  p3320sub0_datatype = 5
  p3320sub0_accesstype = ro
  p3320sub0_pdomapping = 0
  p3320sub1_parametername = ProgIO0.Index
  p3320sub1_objecttype = 7
  p3320sub1_datatype = 6
  p3320sub1_lowlimit = 
  p3320sub1_highlimit = 
  p3320sub1_accesstype = rw
  p3320sub1_pdomapping = 0
  p3320sub1_parametervalue = 
  p3320sub1_objflags = 0
  p3320sub2_parametername = ProgIO0.Subindex
  p3320sub2_objecttype = 7
  p3320sub2_datatype = 6
  p3320sub2_lowlimit = 
  p3320sub2_highlimit = 
  p3320sub2_accesstype = rw
  p3320sub2_pdomapping = 0
  p3320sub2_parametervalue = 
  p3320sub2_objflags = 0
  p3320sub3_parametername = ProgIO0.BitMask
  p3320sub3_objecttype = 7
  p3320sub3_datatype = 7
  p3320sub3_lowlimit = 
  p3320sub3_highlimit = 
  p3320sub3_accesstype = rw
  p3320sub3_pdomapping = 0
  p3320sub3_parametervalue = 
  p3320sub3_objflags = 0
  p3320sub4_parametername = ProgIO0.Switch
  p3320sub4_objecttype = 7
  p3320sub4_datatype = 6
  p3320sub4_lowlimit = 
  p3320sub4_highlimit = 
  p3320sub4_accesstype = rw
  p3320sub4_pdomapping = 0
  p3320sub4_parametervalue = 
  p3320sub4_objflags = 0
  p3320sub5_parametername = ProgIO0.Value1
  p3320sub5_objecttype = 7
  p3320sub5_datatype = 4
  p3320sub5_lowlimit = 
  p3320sub5_highlimit = 
  p3320sub5_accesstype = rw
  p3320sub5_pdomapping = 0
  p3320sub5_parametervalue = 
  p3320sub5_objflags = 0
  p3320sub6_parametername = ProgIO0.Value2
  p3320sub6_objecttype = 7
  p3320sub6_datatype = 4
  p3320sub6_lowlimit = 
  p3320sub6_highlimit = 
  p3320sub6_accesstype = rw
  p3320sub6_pdomapping = 0
  p3320sub6_parametervalue = 
  p3320sub6_objflags = 0
  p3321_parametername = prog io1
  p3321_objecttype = 9
  p3321_subnumber = 0x7
  p3321_parametervalue = 
  p3321_objflags = 0
  p3321sub0_parametername = number of entries
  p3321sub0_objecttype = 7
  p3321sub0_datatype = 5
  p3321sub0_accesstype = ro
  p3321sub0_pdomapping = 0
  p3321sub1_parametername = ProgIO1.Index
  p3321sub1_objecttype = 7
  p3321sub1_datatype = 6
  p3321sub1_lowlimit = 
  p3321sub1_highlimit = 
  p3321sub1_accesstype = rw
  p3321sub1_pdomapping = 0
  p3321sub1_parametervalue = 
  p3321sub1_objflags = 0
  p3321sub2_parametername = ProgIO1.Subindex
  p3321sub2_objecttype = 7
  p3321sub2_datatype = 6
  p3321sub2_lowlimit = 
  p3321sub2_highlimit = 
  p3321sub2_accesstype = rw
  p3321sub2_pdomapping = 0
  p3321sub2_parametervalue = 
  p3321sub2_objflags = 0
  p3321sub3_parametername = ProgIO1.BitMask
  p3321sub3_objecttype = 7
  p3321sub3_datatype = 7
  p3321sub3_lowlimit = 
  p3321sub3_highlimit = 
  p3321sub3_accesstype = rw
  p3321sub3_pdomapping = 0
  p3321sub3_parametervalue = 
  p3321sub3_objflags = 0
  p3321sub4_parametername = ProgIO1.Switch
  p3321sub4_objecttype = 7
  p3321sub4_datatype = 6
  p3321sub4_lowlimit = 
  p3321sub4_highlimit = 
  p3321sub4_accesstype = rw
  p3321sub4_pdomapping = 0
  p3321sub4_parametervalue = 
  p3321sub4_objflags = 0
  p3321sub5_parametername = ProgIO1.Value1
  p3321sub5_objecttype = 7
  p3321sub5_datatype = 4
  p3321sub5_lowlimit = 
  p3321sub5_highlimit = 
  p3321sub5_accesstype = rw
  p3321sub5_pdomapping = 0
  p3321sub5_parametervalue = 
  p3321sub5_objflags = 0
  p3321sub6_parametername = ProgIO1.Value2
  p3321sub6_objecttype = 7
  p3321sub6_datatype = 4
  p3321sub6_lowlimit = 
  p3321sub6_highlimit = 
  p3321sub6_accesstype = rw
  p3321sub6_pdomapping = 0
  p3321sub6_parametervalue = 
  p3321sub6_objflags = 0
  p3322_parametername = prog io2
  p3322_objecttype = 9
  p3322_subnumber = 0x7
  p3322_parametervalue = 
  p3322_objflags = 0
  p3322sub0_parametername = number of entries
  p3322sub0_objecttype = 7
  p3322sub0_datatype = 5
  p3322sub0_accesstype = ro
  p3322sub0_pdomapping = 0
  p3322sub1_parametername = ProgIO2.Index
  p3322sub1_objecttype = 7
  p3322sub1_datatype = 6
  p3322sub1_lowlimit = 
  p3322sub1_highlimit = 
  p3322sub1_accesstype = rw
  p3322sub1_pdomapping = 0
  p3322sub1_parametervalue = 
  p3322sub1_objflags = 0
  p3322sub2_parametername = ProgIO2.Subindex
  p3322sub2_objecttype = 7
  p3322sub2_datatype = 6
  p3322sub2_lowlimit = 
  p3322sub2_highlimit = 
  p3322sub2_accesstype = rw
  p3322sub2_pdomapping = 0
  p3322sub2_parametervalue = 
  p3322sub2_objflags = 0
  p3322sub3_parametername = ProgIO2.BitMask
  p3322sub3_objecttype = 7
  p3322sub3_datatype = 7
  p3322sub3_lowlimit = 
  p3322sub3_highlimit = 
  p3322sub3_accesstype = rw
  p3322sub3_pdomapping = 0
  p3322sub3_parametervalue = 
  p3322sub3_objflags = 0
  p3322sub4_parametername = ProgIO2.Switch
  p3322sub4_objecttype = 7
  p3322sub4_datatype = 6
  p3322sub4_lowlimit = 
  p3322sub4_highlimit = 
  p3322sub4_accesstype = rw
  p3322sub4_pdomapping = 0
  p3322sub4_parametervalue = 
  p3322sub4_objflags = 0
  p3322sub5_parametername = ProgIO2.Value1
  p3322sub5_objecttype = 7
  p3322sub5_datatype = 4
  p3322sub5_lowlimit = 
  p3322sub5_highlimit = 
  p3322sub5_accesstype = rw
  p3322sub5_pdomapping = 0
  p3322sub5_parametervalue = 
  p3322sub5_objflags = 0
  p3322sub6_parametername = ProgIO2.Value2
  p3322sub6_objecttype = 7
  p3322sub6_datatype = 4
  p3322sub6_lowlimit = 
  p3322sub6_highlimit = 
  p3322sub6_accesstype = rw
  p3322sub6_pdomapping = 0
  p3322sub6_parametervalue = 
  p3322sub6_objflags = 0
  p3323_parametername = prog io3
  p3323_objecttype = 9
  p3323_subnumber = 0x7
  p3323_parametervalue = 
  p3323_objflags = 0
  p3323sub0_parametername = number of entries
  p3323sub0_objecttype = 7
  p3323sub0_datatype = 5
  p3323sub0_accesstype = ro
  p3323sub0_pdomapping = 0
  p3323sub1_parametername = ProgIO3.Index
  p3323sub1_objecttype = 7
  p3323sub1_datatype = 6
  p3323sub1_lowlimit = 
  p3323sub1_highlimit = 
  p3323sub1_accesstype = rw
  p3323sub1_pdomapping = 0
  p3323sub1_parametervalue = 
  p3323sub1_objflags = 0
  p3323sub2_parametername = ProgIO3.Subindex
  p3323sub2_objecttype = 7
  p3323sub2_datatype = 6
  p3323sub2_lowlimit = 
  p3323sub2_highlimit = 
  p3323sub2_accesstype = rw
  p3323sub2_pdomapping = 0
  p3323sub2_parametervalue = 
  p3323sub2_objflags = 0
  p3323sub3_parametername = ProgIO3.BitMask
  p3323sub3_objecttype = 7
  p3323sub3_datatype = 7
  p3323sub3_lowlimit = 
  p3323sub3_highlimit = 
  p3323sub3_accesstype = rw
  p3323sub3_pdomapping = 0
  p3323sub3_parametervalue = 
  p3323sub3_objflags = 0
  p3323sub4_parametername = ProgIO3.Switch
  p3323sub4_objecttype = 7
  p3323sub4_datatype = 6
  p3323sub4_lowlimit = 
  p3323sub4_highlimit = 
  p3323sub4_accesstype = rw
  p3323sub4_pdomapping = 0
  p3323sub4_parametervalue = 
  p3323sub4_objflags = 0
  p3323sub5_parametername = ProgIO3.Value1
  p3323sub5_objecttype = 7
  p3323sub5_datatype = 4
  p3323sub5_lowlimit = 
  p3323sub5_highlimit = 
  p3323sub5_accesstype = rw
  p3323sub5_pdomapping = 0
  p3323sub5_parametervalue = 
  p3323sub5_objflags = 0
  p3323sub6_parametername = ProgIO3.Value2
  p3323sub6_objecttype = 7
  p3323sub6_datatype = 4
  p3323sub6_lowlimit = 
  p3323sub6_highlimit = 
  p3323sub6_accesstype = rw
  p3323sub6_pdomapping = 0
  p3323sub6_parametervalue = 
  p3323sub6_objflags = 0
SI_unit_BK1 : FBC.0x00000114.0x00000003.ex250sca1a_v3.0 v3.0 (OrderNumber=SI unit)  [CAN1 -> ILE1F_BK1.CAN2 (NodeNumber=6)]
  pheartbeat_producertime = 1000
  p2000_parametername = Reserved
  p2000_objecttype = 7
  p2000_datatype = 7
  p2000_accesstype = ro
  p2000_pdomapping = 0
  p2001_parametername = Password
  p2001_objecttype = 7
  p2001_datatype = 6
  p2001_accesstype = wo
  p2001_pdomapping = 0
  p2001_parametervalue = 
  p2001_objflags = 0
  p6000_subnumber = 5
  p6000_parametername = Read Input 8Bit
  p6000_objecttype = 8
  p6000_parametervalue = 
  p6000_objflags = 0
  p6000sub0_parametername = Number of Input 8Bit
  p6000sub0_objecttype = 7
  p6000sub0_datatype = 5
  p6000sub0_accesstype = ro
  p6000sub0_pdomapping = 0
  p6100_subnumber = 3
  p6100_parametername = Read Input 16Bit
  p6100_objecttype = 8
  p6100_parametervalue = 
  p6100_objflags = 0
  p6100sub0_parametername = Number of Input 16Bit
  p6100sub0_objecttype = 7
  p6100sub0_datatype = 5
  p6100sub0_accesstype = ro
  p6100sub0_pdomapping = 0
  p6120_subnumber = 2
  p6120_parametername = Read Input 32Bit
  p6120_objecttype = 8
  p6120_parametervalue = 
  p6120_objflags = 0
  p6120sub0_parametername = Number of Input 32Bit
  p6120sub0_objecttype = 7
  p6120sub0_datatype = 5
  p6120sub0_accesstype = ro
  p6120sub0_pdomapping = 0
  p6200_subnumber = 5
  p6200_parametername = Write Output 8Bit
  p6200_objecttype = 8
  p6200_parametervalue = 
  p6200_objflags = 0
  p6200sub0_parametername = Number of Output 8Bit
  p6200sub0_objecttype = 7
  p6200sub0_datatype = 5
  p6200sub0_accesstype = ro
  p6200sub0_pdomapping = 0
  p6206_subnumber = 5
  p6206_parametername = Error Mode Output 8Bit
  p6206_objecttype = 8
  p6206_parametervalue = 
  p6206_objflags = 0
  p6206sub0_parametername = Number of Output 8Bit
  p6206sub0_objecttype = 7
  p6206sub0_datatype = 5
  p6206sub0_accesstype = ro
  p6206sub0_pdomapping = 0
  p6206sub1_parametername = Error Mode Output 1h to 8h
  p6206sub1_objecttype = 7
  p6206sub1_datatype = 5
  p6206sub1_accesstype = rww
  p6206sub1_pdomapping = 0
  p6206sub1_parametervalue = 0xFF
  p6206sub1_objflags = 0
  p6206sub2_parametername = Error Mode Output 9h to 16h
  p6206sub2_objecttype = 7
  p6206sub2_datatype = 5
  p6206sub2_accesstype = rww
  p6206sub2_pdomapping = 0
  p6206sub2_parametervalue = 0xFF
  p6206sub2_objflags = 0
  p6206sub3_parametername = Error Mode Output 17h to 24h
  p6206sub3_objecttype = 7
  p6206sub3_datatype = 5
  p6206sub3_accesstype = rww
  p6206sub3_pdomapping = 0
  p6206sub3_parametervalue = 0xFF
  p6206sub3_objflags = 0
  p6206sub4_parametername = Error Mode Output 25h to 32h
  p6206sub4_objecttype = 7
  p6206sub4_datatype = 5
  p6206sub4_accesstype = rww
  p6206sub4_pdomapping = 0
  p6206sub4_parametervalue = 0xFF
  p6206sub4_objflags = 0
  p6207_subnumber = 5
  p6207_parametername = Error Value Output 8Bit
  p6207_objecttype = 8
  p6207_parametervalue = 
  p6207_objflags = 0
  p6207sub0_parametername = Number of Output 8Bit
  p6207sub0_objecttype = 7
  p6207sub0_datatype = 5
  p6207sub0_accesstype = ro
  p6207sub0_pdomapping = 0
  p6207sub1_parametername = Error Value Output 1h to 8h
  p6207sub1_objecttype = 7
  p6207sub1_datatype = 5
  p6207sub1_accesstype = rw
  p6207sub1_pdomapping = 0
  p6207sub1_parametervalue = 0x00
  p6207sub1_objflags = 0
  p6207sub2_parametername = Error Value Output 9h to 16h
  p6207sub2_objecttype = 7
  p6207sub2_datatype = 5
  p6207sub2_accesstype = rw
  p6207sub2_pdomapping = 0
  p6207sub2_parametervalue = 0x00
  p6207sub2_objflags = 0
  p6207sub3_parametername = Error Value Output 17h to 24h
  p6207sub3_objecttype = 7
  p6207sub3_datatype = 5
  p6207sub3_accesstype = rw
  p6207sub3_pdomapping = 0
  p6207sub3_parametervalue = 0x00
  p6207sub3_objflags = 0
  p6207sub4_parametername = Error Value Output 25h to 32h
  p6207sub4_objecttype = 7
  p6207sub4_datatype = 5
  p6207sub4_accesstype = rw
  p6207sub4_pdomapping = 0
  p6207sub4_parametervalue = 0x00
  p6207sub4_objflags = 0
  p6300_subnumber = 3
  p6300_parametername = Write Output 16Bit
  p6300_objecttype = 8
  p6300_parametervalue = 
  p6300_objflags = 0
  p6300sub0_parametername = Number of Output 16Bit
  p6300sub0_objecttype = 7
  p6300sub0_datatype = 5
  p6300sub0_accesstype = ro
  p6300sub0_pdomapping = 0
  p6306_subnumber = 3
  p6306_parametername = Error Mode Output 16Bit
  p6306_objecttype = 8
  p6306_parametervalue = 
  p6306_objflags = 0
  p6306sub0_parametername = Number of Output 16Bit
  p6306sub0_objecttype = 7
  p6306sub0_datatype = 5
  p6306sub0_accesstype = ro
  p6306sub0_pdomapping = 0
  p6306sub1_parametername = Error Mode Output 1h to 16h
  p6306sub1_objecttype = 7
  p6306sub1_datatype = 6
  p6306sub1_accesstype = rww
  p6306sub1_pdomapping = 0
  p6306sub1_parametervalue = 0xFFFF
  p6306sub1_objflags = 0
  p6306sub2_parametername = Error Mode Output 17h to 32h
  p6306sub2_objecttype = 7
  p6306sub2_datatype = 6
  p6306sub2_accesstype = rww
  p6306sub2_pdomapping = 0
  p6306sub2_parametervalue = 0xFFFF
  p6306sub2_objflags = 0
  p6307_subnumber = 3
  p6307_parametername = Error Value Output 16Bit
  p6307_objecttype = 8
  p6307_parametervalue = 
  p6307_objflags = 0
  p6307sub0_parametername = Number of Output 16Bit
  p6307sub0_objecttype = 7
  p6307sub0_datatype = 5
  p6307sub0_accesstype = ro
  p6307sub0_pdomapping = 0
  p6307sub1_parametername = Error Value Output 1h to 16h
  p6307sub1_objecttype = 7
  p6307sub1_datatype = 6
  p6307sub1_accesstype = rw
  p6307sub1_pdomapping = 0
  p6307sub1_parametervalue = 0x0000
  p6307sub1_objflags = 0
  p6307sub2_parametername = Error Value Output 17h to 32h
  p6307sub2_objecttype = 7
  p6307sub2_datatype = 6
  p6307sub2_accesstype = rw
  p6307sub2_pdomapping = 0
  p6307sub2_parametervalue = 0x0000
  p6307sub2_objflags = 0
  p6320_subnumber = 2
  p6320_parametername = Write Output 32Bit
  p6320_objecttype = 8
  p6320_parametervalue = 
  p6320_objflags = 0
  p6320sub0_parametername = Number of Output 32Bit
  p6320sub0_objecttype = 7
  p6320sub0_datatype = 5
  p6320sub0_accesstype = ro
  p6320sub0_pdomapping = 0
  p6326_subnumber = 2
  p6326_parametername = Error Mode Output 32Bit
  p6326_objecttype = 8
  p6326_parametervalue = 
  p6326_objflags = 0
  p6326sub0_parametername = Number of Output 32Bit
  p6326sub0_objecttype = 7
  p6326sub0_datatype = 5
  p6326sub0_accesstype = ro
  p6326sub0_pdomapping = 0
  p6326sub1_parametername = Error Mode Output 1h to 32h
  p6326sub1_objecttype = 7
  p6326sub1_datatype = 7
  p6326sub1_accesstype = rww
  p6326sub1_pdomapping = 0
  p6326sub1_parametervalue = 0xFFFFFFFF
  p6326sub1_objflags = 0
  p6327_subnumber = 2
  p6327_parametername = Error Value Output 32Bit
  p6327_objecttype = 8
  p6327_parametervalue = 
  p6327_objflags = 0
  p6327sub0_parametername = Number of Output 32Bit
  p6327sub0_objecttype = 7
  p6327sub0_datatype = 5
  p6327sub0_accesstype = ro
  p6327sub0_pdomapping = 0
  p6327sub1_parametername = Error Value Output 1h to 32h
  p6327sub1_objecttype = 7
  p6327sub1_datatype = 7
  p6327sub1_accesstype = rw
  p6327sub1_pdomapping = 0
  p6327sub1_parametervalue = 0x00000000
  p6327sub1_objflags = 0
X20AI4322_008 : X20AI4322 v1.2.0.0  [SS1 -> X20TB12a.SS; SL -> X20BM11e.SL1]
  LowerLimit = -8000
  ChannelType01 = 4 to 20mA
  ChannelType02 = 4 to 20mA
  ChannelType03 = 4 to 20mA
  ChannelType04 = 4 to 20mA
X20AO4622_009 : X20AO4622 v1.3.0.0  [SS1 -> X20TB12c.SS; SL -> X20BM11h.SL1]
X20AT4222_010 : X20AT4222 v1.4.0.0  [SS1 -> X20TB12b.SS; SL -> X20BM11g.SL1]
X20BM01 : X20BM01 v2.2.0.0  [X2X1 -> X20BM11d.X2X2]
X20BM11 : X20BM11 v1.1.0.0  [X2X1 -> X20CP1382.IF6]
X20BM11a : X20BM11 v1.1.0.0  [X2X1 -> X20BM11.X2X2]
X20BM11b : X20BM11 v1.1.0.0  [X2X1 -> X20BM11a.X2X2]
X20BM11c : X20BM11 v1.1.0.0  [X2X1 -> X20BM11b.X2X2]
X20BM11d : X20BM11 v1.1.0.0  [X2X1 -> X20BM11v.X2X2]
X20BM11e : X20BM11 v1.1.0.0  [X2X1 -> X20BM01.X2X2]
X20BM11g : X20BM11 v1.1.0.0  [X2X1 -> X20BM11h.X2X2]
X20BM11h : X20BM11 v1.1.0.0  [X2X1 -> X20BM11e.X2X2]
X20BM11v : X20BM11 v1.1.0.0  [X2X1 -> X20BM11c.X2X2]
X20BM31 : X20BM31 v1.1.0.0  [X2X1 -> X20BM11g.X2X2]
X20BM31a : X20BM31 v1.1.0.0  [X2X1 -> X20BM31.X2X2]
X20CP1382 : X20CP1382 v1.14.0.0  [X1 -> X1.SL; X2 -> X2.SL; X3 -> X3.SL]
  Module X1 (Type=X1, Virtual=true, Version=1.14.0.0)
    Connection (Connector=SS1, TargetModule=X20TB1F, TargetConnector=SS)
    Connection (Connector=SL, TargetModule=X20CP1382, TargetConnector=X1)
  Module X2 (Type=X2, Virtual=true, Version=1.14.0.0)
    Connection (Connector=SS1, TargetModule=X20TB1F1, TargetConnector=SS)
    Connection (Connector=SL, TargetModule=X20CP1382, TargetConnector=X2)
  Module X3 (Type=X3, Virtual=true, Version=1.14.0.0)
    Connection (Connector=SS1, TargetModule=X20TB1F2, TargetConnector=SS)
    Connection (Connector=SL, TargetModule=X20CP1382, TargetConnector=X3)
    X3Channel05Config = input
    X3Channel06Config = input
    X3Channel07Config = input
  Connector IF2:
    ActivateDevice = 1
    Mode = Manual
    InternetAddress = 192.168.127.10
    SubnetMask = 255.255.255.0
    InaNodeNumber = 0
  Connector IF3:
    MtuSize = 1000
    DNAConfiguration = manual
    CycleTime = 2000
  Connector IF7:
    Baudrate = 250000
    ActivateCANIO = 0
    ActivateCanOpen = 1
    pnmtstartup_maximumbootuptime = 15
    pnmtstartup_pnptimer = 1
    procPriority = 197
    pheartbeat_producertime = 0
    pheartbeat_securityfactor = 0
    pactivatesync = 1
    pcycleperiod = 10000
    pwindowlength = 10000
    p1006_parametervalue = 0
    p1007_parametervalue = 0
    p100c_parametervalue = 1000
    p100d_parametervalue = 3
  ConfigurationID = 1BK2Bar
  ConfigVersion = 1.0.1
  UserPartitionSize = 400
  PermanentPvSize = 25000
  RemanentGlobalPvSize = 5000
  VolatileGlobalPvSize = 300000
  UserLoggerSize = 4096000
  EnableUsbRemoteInstall = 1
  EnableCfRemoteInstall = 1
  TimerDeviceType = EPLX2X
  TimerDevice = X20CP1382.IF3
  IdleTaskClass = 3
  TaskClassIdleTime = 8000
  Cyclic1Duration = 4000  // In this Cyclic task is located Stepper by X2X commns
  Cyclic1Tolerance = 0
  Cyclic1Stack = 16000
  Cyclic1Output = 1
  Cyclic2Duration = 12000
  Cyclic2Tolerance = 0
  Cyclic3Duration = 16000
  Cyclic3Tolerance = 16000
  Cyclic4Duration = 32000
  Cyclic4Tolerance = 32000
  Cyclic5Duration = 80000
  Cyclic5Tolerance = 80000
  Cyclic6Duration = 88000
  Cyclic6Tolerance = 88000
  Cyclic7Duration = 44000
  Cyclic7Tolerance = 88000
  Cyclic8Duration = 200000
  TimeZone = 150
  ActivateDaylightSavingTime = 1
  FtpUser1
  FtpUsername1 = EFI  // EFI
  FtpUserPassword1 = G25QVEacZZSwxmUMISDzqyniZhuiJFyYu3vry1aXZ8A=  // Castellon
  FtpUserSalt1 = u5fK9ZrP
  FTPAccessRight1 = 0
X20DIF371_001 : X20DIF371 v1.3.0.0  [SS1 -> X20TB1F3.SS; SL -> X20BM11.SL1]
  Supervision = off
X20DIF371_002 : X20DIF371 v1.3.0.0  [SS1 -> X20TB1F4.SS; SL -> X20BM11a.SL1]
  Supervision = off
X20DIF371_003 : X20DIF371 v1.3.0.0  [SS1 -> X20TB1F5.SS; SL -> X20BM11b.SL1]
  Supervision = off
X20DIF371_004 : X20DIF371 v1.3.0.0  [SS1 -> X20TB1F6.SS; SL -> X20BM11c.SL1]
  Supervision = off
X20DOF322_005 : X20DOF322 v1.5.0.0  [SS1 -> X20TB1F24.SS; SL -> X20BM11v.SL1]
  Supervision = off
X20DOF322_006 : X20DOF322 v1.5.0.0  [SS1 -> X20TB1F25.SS; SL -> X20BM11d.SL1]
  Supervision = off
X20PS3300_007 : X20PS3300 v1.4.0.0  [SS1 -> X20TB12.SS; SL -> X20BM01.SL1]
X20SM1436_011 : X20SM1436 v2.3.0.0  [SS1 -> X20TB12u.SS; SL -> X20BM31.SL1]
  Supervision = off
  DelayedCurrentSwitchOff01 = 5
  HoldingCurrent = 30
  RatedCurrent = 100
  MaximumCurrent = 110
  SM_SCALE_STEP_r1 = 100
X20SM1436_012 : X20SM1436 v2.3.0.0  [SS1 -> X20TB12v.SS; SL -> X20BM31a.SL1]
  Supervision = off
  DelayedCurrentSwitchOff01 = 5
  HoldingCurrent = 30
  RatedCurrent = 100
  MaximumCurrent = 110
  SM_SCALE_STEP_r1 = 100
X20TB12 : X20TB12 v1.0.0.0
X20TB12a : X20TB12 v1.0.0.0
X20TB12b : X20TB12 v1.0.0.0
X20TB12c : X20TB12 v1.0.0.0
X20TB12u : X20TB12 v1.0.0.0
X20TB12v : X20TB12 v1.0.0.0
X20TB1F : X20TB1F v1.0.0.0
X20TB1F1 : X20TB1F v1.0.0.0
X20TB1F2 : X20TB1F v1.0.0.0
X20TB1F24 : X20TB1F v1.0.0.0
X20TB1F25 : X20TB1F v1.0.0.0
X20TB1F3 : X20TB1F v1.0.0.0
X20TB1F4 : X20TB1F v1.0.0.0
X20TB1F5 : X20TB1F v1.0.0.0
X20TB1F6 : X20TB1F v1.0.0.0
```

### Cpu.per - X20CP1382/Cpu.per
```iecst
VAR_CONFIG
	gPermanentSN AT %M0; (*Serial Number of the machine*)
	gPermanentVersion AT %M100; (* *)
	gPermanentMachine AT %M148; (* *)
	gPermanentSwBelt AT %M500; (* *)
	gPermanentBlock AT %M600; (* *)
	gPermanentInksParSw AT %M800; (* *)
	gInksPermanentParBar AT %M2600; (* *)
	HoldingRegister AT %MW6000; (* *)
END_VAR
```

### .gitignore - X20CP1382/EFI/.gitignore
```
BusNavigator.xostd
```

### EVENT.MEV - X20CP1382/EFI/EVENT.MEV
```
1500448763	60010000	sainz-penal	2	1	SafeMODULE ID
1500448764	60010000	sainz-penal	2	2	SafeMODULE ID
1500448765	60010000	sainz-penal	2	3	SafeMODULE ID
1500448766	60010000	sainz-penal	2	4	SafeMODULE ID
1500448767	60010000	sainz-penal	2	5	SafeMODULE ID
1500448768	60010000	sainz-penal	2	6	SafeMODULE ID
1500448769	60020000	sainz-penal	3	1	X20SLX402	SafeMODULE ID
1500448770	60020000	sainz-penal	3	2	X20SI2100	SafeMODULE ID
1500448771	60020000	sainz-penal	3	3	X20SI8110	SafeMODULE ID
1500448772	60020000	sainz-penal	3	4	X20SO2110	SafeMODULE ID
1500448773	60020000	sainz-penal	3	5	X20SI8110	SafeMODULE ID
1500448774	60020000	sainz-penal	3	6	X20SO2110	SafeMODULE ID
1500448874	30010000	sainz-penal	2	Variables:Main	85C07E2B
1500448932	20040000	sainz-penal	1	A97AF89C
1500449013	30010000	sainz-penal	2	Variables:Main	EDA1E9ED
1500449296	20040000	sainz-penal	1	74DCC96B
1500449314	30010000	sainz-penal	2	Variables:Main	20453E72
1500449482	20040000	sainz-penal	1	41AB98BF
1500449505	30020000	sainz-penal	2	Code:Main	17411027
1500449512	20050000	sainz-penal	2	9E945EA8	6B9BCED3
1500449552	20040000	sainz-penal	1	6D0A151A
1500449570	30020000	sainz-penal	2	Code:Main	3612C10B
1500449575	20050000	sainz-penal	2	E5B10D58	C9E42BB4
1500460549	30020000	sainz-penal	2	Code:Main	FEB6A290
1500460910	20040000	sainz-penal	1	B86A12DA
1500461071	20040000	sainz-penal	1	D214E2F9
1500461932	20040000	sainz-penal	1	27152325
1500461940	20040000	sainz-penal	1	D214E2F9
1500461972	20040000	sainz-penal	1	B76968BB
1500462529	20040000	sainz-penal	1	4D4BE879
1500462696	30020000	sainz-penal	2	Code:Main	7E137E14
1500462818	20040000	sainz-penal	1	EAF1ED23
1500462875	30020000	sainz-penal	2	Code:Main	8B6AC711
1500463401	30020000	sainz-penal	2	Code:Main	216FB661
1500463624	20040000	sainz-penal	1	4D4BE879
1500464015	20040000	sainz-penal	1	2E4BC1D2
1500464043	30020000	sainz-penal	2	Code:Main	108B1069
1500464075	20040000	sainz-penal	1	1EBF861E
1500464081	30020000	sainz-penal	2	Code:Main	7AC26481
1500477228	30010000	sainz-penal	2	Variables:Main	C5D89750
1500477380	30020000	sainz-penal	2	Code:Main	8253F9DB
1500477389	30020000	sainz-penal	2	Code:Main	B704E02A
1500477473	30020000	sainz-penal	2	Code:Main	E3FD2E08
1500477695	30020000	sainz-penal	2	Code:Main	4A8FCE2B
1500477748	30020000	sainz-penal	2	Code:Main	8FF91979
1500477943	30020000	sainz-penal	2	Code:Main	34DC030F
1500478096	30020000	sainz-penal	2	Code:Main	818A5EDD
1500478109	30010000	sainz-penal	2	Variables:Main	10794F87
1500478126	30010000	sainz-penal	2	Variables:Main	E7FCDF7B
1500478157	30010000	sainz-penal	2	Variables:Main	FAA753E5
1500478233	30020000	sainz-penal	2	Code:Main	7FA10A5E
1500478420	30020000	sainz-penal	2	Code:Main	299956DD
1500478421	20040000	sainz-penal	1	450E4729
1500478446	30020000	sainz-penal	2	Code:Main	C263F3B4
1500478526	20040000	sainz-penal	1	D24DDF80
1500478774	30010000	sainz-penal	2	Variables:Main	9ADCF77A
1500478842	30020000	sainz-penal	2	Code:Main	E2A077CC
1500478869	20040000	sainz-penal	1	A404BB33
1500478907	20040000	sainz-penal	1	D24DDF80
1500479059	30020000	sainz-penal	2	Code:Main	070A4C3C
1500479156	30010000	sainz-penal	2	Variables:Main	FAA753E5
1500479206	30020000	sainz-penal	2	Code:Main	A5724779
1500479245	20040000	sainz-penal	1	57DCDBAB
1500479297	20040000	sainz-penal	1	B0A6844F
1500479342	20040000	sainz-penal	1	0F68F1F6
1500479501	30020000	sainz-penal	2	Code:Main	77990BCD
1500479521	30020000	sainz-penal	2	Code:Main	F644283C
1500479608	30020000	sainz-penal	2	Code:Main	99211326
1500479996	30010000	sainz-penal	2	Variables:MOVE_INT	FCBFCD51
1500479997	30030000	sainz-penal	1	MOVE_INT
1500480077	30010000	sainz-penal	2	Variables:MOVE_INT	1F84B4A9
1500480093	30020000	sainz-penal	2	MOVE_INT:MOVE_INT	516DB6CA
1500480184	30010000	sainz-penal	2	Variables:Main	56E2DC78
1500480236	30020000	sainz-penal	2	Code:Main	FCC3E2A1
1500480252	30020000	sainz-penal	2	Code:Main	4F76F181
1500480264	30020000	sainz-penal	2	Code:Main	FCC3E2A1
1500480285	30010000	sainz-penal	2	Variables:Main	667160D7
1500480297	30020000	sainz-penal	2	Code:Main	FBBC8861
1500480427	30020000	sainz-penal	2	Code:Main	3D02AD94
1500480642	30020000	sainz-penal	2	Code:Main	BBFF8770
1500480665	30020000	sainz-penal	2	Code:Main	F542FFC0
1500480788	30020000	sainz-penal	2	Code:Main	5052D2C0
1500480980	30010000	sainz-penal	2	Variables:Main	65757759
1500481045	30020000	sainz-penal	2	Code:Main	B9AD912C
1500481126	30010000	sainz-penal	2	Variables:Main	C544F49E
1500481144	30020000	sainz-penal	2	Code:Main	25A48754
1500481369	30020000	sainz-penal	2	Code:Main	D1E7356B
1500481386	20040000	sainz-penal	1	5EA12F1B
1500481404	20040000	sainz-penal	1	022EAA0A
1500481418	30020000	sainz-penal	2	Code:Main	521D4C0D
1500481459	20040000	sainz-penal	1	010AE2BA
1500481477	20040000	sainz-penal	1	B4B6EDCC
1500481498	30020000	sainz-penal	2	Code:Main	B8923760
1500481660	30020000	sainz-penal	2	Code:Main	BB7F1456
1500481672	20050000	sainz-penal	2	F33927EB	2A387214
1500482936	30020000	sainz-penal	2	Code:Main	95860917
1500495749	20040000	sainz-penal	1	C4CE020F
1500495989	30020000	sainz-penal	2	Code:Main	781B249A
1500496062	20040000	sainz-penal	1	94986B59
1500496073	30020000	sainz-penal	2	Code:Main	1CB81FDE
1500496109	30040000	sainz-penal	1	MOVE_INT
1500496126	30010000	sainz-penal	2	Variables:Main	7684D8F0
1500496133	20050000	sainz-penal	2	178289DD	3FA7ACCF
1500496951	20040000	sainz-penal	1	744F4B30
1500496968	30020000	sainz-penal	2	Code:Main	B4AC970E
1500497307	30020000	sainz-penal	2	Code:Main	7ED35F23
1500497469	30020000	sainz-penal	2	Code:Main	AB793EE0
1500497477	20050000	sainz-penal	2	8530A4D8	B6837389
1500497539	30020000	sainz-penal	2	Code:Main	17225637
1500497546	20050000	sainz-penal	2	189EF542	C44B20F2
1500497899	30020000	sainz-penal	2	Code:Main	E54CF4E4
1500498091	20040000	sainz-penal	1	FDF14932
1500498107	20040000	sainz-penal	1	446AA030
1500498113	30020000	sainz-penal	2	Code:Main	6229C055
1500498120	20050000	sainz-penal	2	F36BAB27	27FC5ED4
1500498639	30010000	sainz-penal	2	Variables:MOVE_UINT	FCBFCD51
1500498640	30030000	sainz-penal	1	MOVE_UINT
1500498684	30010000	sainz-penal	2	Variables:MOVE_UINT	D5C16BB2
1500498696	30020000	sainz-penal	2	MOVE_UINT:MOVE_UINT	B19BD614
1500498701	30020000	sainz-penal	2	Code:Main	992896CD
1500498714	30020000	sainz-penal	2	Code:Main	E640EDB9
1500498789	30010000	sainz-penal	2	Variables:MOVE_UINT	16499C79
1500498797	20050000	sainz-penal	2	F36BAB27	27FC5ED4
1500498823	20040000	sainz-penal	1	CB8F5E9A
1500498859	20040000	sainz-penal	1	D1999B16
1500498951	30010000	sainz-penal	2	Variables:MOVE_UINT	09D85549
1500498967	30020000	sainz-penal	2	Code:Main	D7544315
1500498968	20040000	sainz-penal	1	73A6888A
1500498976	30020000	sainz-penal	2	Code:Main	E640EDB9
1500498984	20050000	sainz-penal	2	F36BAB27	27FC5ED4
1500498999	30020000	sainz-penal	2	MOVE_UINT:MOVE_UINT	93DAC6D9
1500499020	30020000	sainz-penal	2	MOVE_UINT:MOVE_UINT	7D1DE0EA
1500499053	30020000	sainz-penal	2	MOVE_UINT:MOVE_UINT	D8ED5AB7
1500499063	30020000	sainz-penal	2	MOVE_UINT:MOVE_UINT	ADD2C97D
1500499075	30020000	sainz-penal	2	MOVE_UINT:MOVE_UINT	D8ED5AB7
1500499128	30020000	sainz-penal	2	MOVE_UINT:MOVE_UINT	953385FF
1500499151	30020000	sainz-penal	2	MOVE_UINT:MOVE_UINT	01BA0DB0
1500499174	30020000	sainz-penal	2	MOVE_UINT:MOVE_UINT	953385FF
1500499225	30020000	sainz-penal	2	MOVE_UINT:MOVE_UINT	B78771D9
1500499245	30020000	sainz-penal	2	MOVE_UINT:MOVE_UINT	6434322A
1500499281	30010000	sainz-penal	2	Variables:MOVE_UINT	24C94126
1500499302	30020000	sainz-penal	2	MOVE_UINT:MOVE_UINT	2A89D4C3
1500499311	30020000	sainz-penal	2	MOVE_UINT:MOVE_UINT	0E62EA16
1500499318	30020000	sainz-penal	2	MOVE_UINT:MOVE_UINT	C3B3FF8F
1500499325	20050000	sainz-penal	2	F36BAB27	27FC5ED4
1500499497	30020000	sainz-penal	2	MOVE_UINT:MOVE_UINT	D592E5C8
1500499506	20050000	sainz-penal	2	F36BAB27	27FC5ED4
1500499515	30020000	sainz-penal	2	MOVE_UINT:MOVE_UINT	34156FAD
1500499518	30010000	sainz-penal	2	Variables:MOVE_UINT	09D85549
1500499527	20050000	sainz-penal	2	F36BAB27	27FC5ED4
1500499574	30010000	sainz-penal	2	Variables:Main	D1D07E99
1500499609	30010000	sainz-penal	2	Variables:MOVE_UINT	0D9D90F6
1500499611	30020000	sainz-penal	2	Code:Main	1131BF33
1500499623	30020000	sainz-penal	2	Code:Main	E640EDB9
1500499638	30010000	sainz-penal	2	Variables:Main	7684D8F0
1500499645	20050000	sainz-penal	2	F36BAB27	27FC5ED4
1500499661	30010000	sainz-penal	2	Variables:Main	A6D74E0F
1500499736	20040000	sainz-penal	1	CC2441EF
1500499742	30020000	sainz-penal	2	Code:Main	30F20C51
1500499783	20040000	sainz-penal	1	0C6E9511
1500499825	30020000	sainz-penal	2	Code:Main	0AFECD27
1500499877	30010000	sainz-penal	2	Variables:MOVE_UINT	33B4DA77
1500499902	20050000	sainz-penal	2	60621821	DF3BC896
1500499947	20040000	sainz-penal	1	92166070
1500499967	30010000	sainz-penal	2	Variables:Main	C8361B7F
1500499997	30020000	sainz-penal	2	Code:Main	AC1CA732
1500500006	20050000	sainz-penal	2	593CCCEA	F4F9AB88
1500500208	20040000	sainz-penal	1	72DB0B81
1500500251	30020000	sainz-penal	2	Code:Main	E043CBE8
1500500272	30010000	sainz-penal	2	Variables:Main	DDDEE151
1500500301	30020000	sainz-penal	2	Code:Main	7E493FB6
1500500504	30010000	sainz-penal	2	Variables:MOVE_UINT	4498B2E9
1500500657	30020000	sainz-penal	2	MOVE_UINT:MOVE_UINT	84FBD745
1500500663	30020000	sainz-penal	2	Code:Main	C400487E
1500500681	30020000	sainz-penal	2	MOVE_UINT:MOVE_UINT	2C41593A
1500500689	30020000	sainz-penal	2	Code:Main	D35CDDEE
1500500705	30010000	sainz-penal	2	Variables:Main	7684D8F0
1500500714	20050000	sainz-penal	2	BDC37565	0C1E7337
1500500731	30010000	sainz-penal	2	Variables:Main	D86632B2
1500500764	30020000	sainz-penal	2	Code:Main	006DE174
1500500772	20050000	sainz-penal	2	17857978	486F2BB3
1500500913	20050000	sainz-penal	2	17857978	486F2BB3
1500531159	30010000	sainz-penal	2	Variables:Main	7F60B3B3
1500531284	30010000	sainz-penal	2	Variables:Main	AC84EAEA
1500531455	20040000	sainz-penal	1	CBCD03BE
1500531528	20040000	sainz-penal	1	2236C303
1500531630	30010000	sainz-penal	2	Variables:Main	0ACC24A9
1500532220	30020000	sainz-penal	2	Code:Main	2CAAE795
1500532341	30020000	sainz-penal	2	Code:Main	549D55A7
1500532385	30020000	sainz-penal	2	Code:Main	86E8F8EA
1500532409	30010000	sainz-penal	2	Variables:Main	645D852B
1500532441	30010000	sainz-penal	2	Variables:Main	52CABF21
1500532448	30020000	sainz-penal	2	Code:Main	6DB63C2B
1500532477	30010000	sainz-penal	2	Variables:Main	8E40A5EE
1500533034	30020000	sainz-penal	2	Code:Main	BD9DFBE6
1500533045	30010000	sainz-penal	2	Variables:Main	E6838EE2
1500533053	20050000	sainz-penal	2	FE2A9C87	AD2D9C9F
1500533238	30010000	sainz-penal	2	Variables:Main	9720DF8F
1500533271	30020000	sainz-penal	2	Code:Main	6E0CFD2F
1500533295	20040000	sainz-penal	1	72733D79
1500533332	20040000	sainz-penal	1	746A6088
1500533371	30010000	sainz-penal	2	Variables:Main	5B01BEF1
1500533391	30020000	sainz-penal	2	Code:Main	F91D9412
1500533413	30020000	sainz-penal	2	Code:Main	F66C42B4
1500533421	20050000	sainz-penal	2	D1F76062	EA4A0448
1500533545	30020000	sainz-penal	2	Code:Main	29E55B15
1500533603	30010000	sainz-penal	2	Variables:Main	526B4A5B
1500533753	30010000	sainz-penal	2	Variables:Main	DBE1EC25
1500533819	20040000	sainz-penal	1	D4C9DFEB
1500533829	20040000	sainz-penal	1	AC2DC575
1500533873	30010000	sainz-penal	2	Variables:Main	9977F321
1500533899	30010000	sainz-penal	2	Variables:Main	7F607AA0
1500533950	30010000	sainz-penal	2	Variables:Main	BB380191
1500533963	30020000	sainz-penal	2	Code:Main	AD05E061
1500533973	20050000	sainz-penal	2	63890914	52A816BE
1500534041	20050000	sainz-penal	2	63890914	52A816BE
1500534102	30010000	sainz-penal	2	Variables:Main	14C3AF1A
1500534135	20040000	sainz-penal	1	A4A72A53
1500534159	30010000	sainz-penal	2	Variables:Main	6C8CBA0B
1500534255	30010000	sainz-penal	2	Variables:Main	85F56E99
1500534403	30020000	sainz-penal	2	Code:Main	81A8A527
1500534431	20040000	sainz-penal	1	D0D17531
1500534435	30020000	sainz-penal	2	Code:Main	16B70DEF
1500534443	20050000	sainz-penal	2	1B92D6A2	8CDE713D
1500534475	20040000	sainz-penal	1	80D6ED32
1500534538	30020000	sainz-penal	2	Code:Main	888D623A
1500534548	20050000	sainz-penal	2	35F5266A	1224B691
1500536803	30020000	sainz-penal	2	Code:Main	1C936A19
1500536810	20050000	sainz-penal	2	6375AAEB	4E0658DC
1500536878	20040000	sainz-penal	1	CC079D4E
1500536994	30020000	sainz-penal	2	Code:Main	853CC802
1500537002	20050000	sainz-penal	2	B3FC4148	1503E89A
1500537621	30020000	sainz-penal	2	Code:Main	AD2BA24A
1500537629	20050000	sainz-penal	2	583073F0	44E269CF
1500544273	20040000	sainz-penal	1	2AC61D8F
1500544371	20040000	sainz-penal	1	68784CFE
1500544408	30020000	sainz-penal	2	Code:Main	D564718D
1500544430	30010000	sainz-penal	2	Variables:Main	4221F908
1500544468	30010000	sainz-penal	2	Variables:Main	1F5D8439
1500544486	30020000	sainz-penal	2	Code:Main	26FC4CE2
1500544529	60010000	sainz-penal	2	1	SafeMODULE ID
1500544543	20050000	sainz-penal	2	B820991C	6C77C767
1500545181	20050000	sainz-penal	2	B820991C	6C77C767
1500548053	60010000	sainz-penal	2	1	SafeMODULE ID
1500548069	20050000	sainz-penal	2	DEB8A659	6C77C767
1500550498	60010000	sainz-penal	2	1	SafeMODULE ID
1500550506	20050000	sainz-penal	2	B820991C	6C77C767
1501075023	30010000	sainz-penal	2	Variables:Main	6E8D534D
1501075095	30010000	sainz-penal	2	Variables:Main	9EDE86D9
1501075176	30020000	sainz-penal	2	Code:Main	8BC13812
1501075200	20040000	sainz-penal	1	D0E89A6C
1501075209	20050000	sainz-penal	2	25B8BD67	D6296E20
1501075273	30020000	sainz-penal	2	Code:Main	DCD6DBEE
1501075282	20050000	sainz-penal	2	EB770A78	8E2A1E50
1501075457	30020000	sainz-penal	2	Code:Main	B17D9085
1501077852	30020000	sainz-penal	2	Code:Main	011C3A88
1501077894	30010000	sainz-penal	2	Variables:MOVE_UINT	D1240E3C
1501078098	30020000	sainz-penal	2	MOVE_UINT:MOVE_UINT	34344219
1501078099	30020000	sainz-penal	2	Code:Main	25B5C80A
1501078195	30020000	sainz-penal	2	MOVE_UINT:MOVE_UINT	56316585
1501078243	30020000	sainz-penal	2	MOVE_UINT:MOVE_UINT	F6E765DF
1501078388	30020000	sainz-penal	2	Code:Main	61C9AF2E
1501078400	20040000	sainz-penal	1	1F77CAF0
1501078405	30020000	sainz-penal	2	Code:Main	06C69381
1501078437	30010000	sainz-penal	2	Variables:Main	E110BCA9
1501078447	20050000	sainz-penal	2	D00CBEC8	F87E0A61
1501078621	30020000	sainz-penal	2	MOVE_UINT:MOVE_UINT	93097672
1501078632	30010000	sainz-penal	2	Variables:Main	590E912F
1501078641	20050000	sainz-penal	2	826B2E30	723A687A
1501078984	20050000	sainz-penal	2	826B2E30	723A687A
1501080464	20040000	IVAN	1	EBF94179
1501080537	20040000	IVAN	1	40A784A8
1501080550	20050000	IVAN	2	7F44D19D	601008AC
1501080881	20040000	IVAN	1	67ADF879
1501080908	20040000	IVAN	1	E69F3D84
1501080989	20040000	IVAN	1	02010FB1
1501081071	20040000	IVAN	1	459579FF
1501081088	20040000	IVAN	1	01EB5C84
1501081110	20040000	IVAN	1	D4BA33D6
1501081185	20040000	IVAN	1	D2E82BAE
1501081507	20040000	IVAN	1	328BF2E9
1501081602	20040000	IVAN	1	750BDFB1
1501081619	20040000	IVAN	1	C639C998
1501081658	20040000	IVAN	1	18EB827D
1501081680	20040000	IVAN	1	91AE39AC
1501081953	20040000	IVAN	1	BD7CD8DF
1501081990	20040000	IVAN	1	3B5E7161
1501082198	30020000	IVAN	2	Code:Main	65AC6BF8
1501082214	20040000	IVAN	1	13E1B3F4
1501082398	30010000	IVAN	2	Variables:Main	D0E185B4
1501082620	30010000	IVAN	2	Variables:Main	48758A92
1501082643	20040000	IVAN	1	1DC177F8
1501082893	20040000	IVAN	1	1C1CAB82
1501082924	20040000	IVAN	1	FCCA72C8
1501082945	20040000	IVAN	1	5EF80097
1501082980	30020000	IVAN	2	Code:Main	F3FEE77D
1501083104	30020000	IVAN	2	Code:Main	C8B61F3E
1501083148	30010000	IVAN	2	Variables:Main	2E2EF792
1501083180	30010000	IVAN	2	Variables:Main	CE79C166
1501083192	30020000	IVAN	2	Code:Main	6C87FCE9
1501083214	30010000	IVAN	2	Variables:Main	E2AC1BCE
1501083336	60010000	IVAN	2	1	SafeMODULE ID
1501083346	20050000	IVAN	2	4B79C7EF	3CDFDD09
1501083542	60010000	IVAN	2	1	SafeMODULE ID
1501083731	60010000	IVAN	2	3	SafeMODULE ID
1501083780	20050000	IVAN	2	A824E1B2	3CDFDD09
1501085234	20050000	IVAN	2	A824E1B2	3CDFDD09
1501085649	20050000	IVAN	2	A824E1B2	3CDFDD09
1501140074	20050000	IVAN	2	A824E1B2	3CDFDD09
1501141028	60010000	IVAN	2	1	SafeMODULE ID
1501141040	20050000	IVAN	2	4F9B300A	3CDFDD09
1501151021	70010100	IVAN	1	-if tcpip -ip 10.138.82.22 -p 50000
1501151769	60010000	IVAN	2	1	SafeMODULE ID
1501151788	20050000	IVAN	2	EDB3BD59	3CDFDD09
1501151831	60010000	IVAN	2	2	SafeMODULE ID
1501151861	60010000	IVAN	2	3	SafeMODULE ID
1501151868	60010000	IVAN	2	4	SafeMODULE ID
1501151890	20050000	IVAN	2	593F5045	3CDFDD09
1501167655	30020000	IVAN	2	Code:Main	8222BA45
1501167671	20050000	IVAN	2	088D9E82	DC1973C1
1501168150	60010000	IVAN	2	3	SafeMODULE ID
1501168164	20050000	IVAN	2	877BEFA1	DC1973C1
1501168220	60010000	IVAN	2	3	SafeMODULE ID
1501168320	60010000	IVAN	2	3	SafeMODULE ID
1501168370	60010000	IVAN	2	3	SafeMODULE ID
1501168481	20050000	IVAN	2	088D9E82	DC1973C1
1501168510	60010000	IVAN	2	3	SafeMODULE ID
1501168595	20050000	IVAN	2	5C335F15	DC1973C1
1501169365	30020000	IVAN	2	Code:Main	605670EE
1501169384	20050000	IVAN	2	542AC7CC	797A1D80
1501169735	30020000	IVAN	2	Code:Main	0B626BEE
1501169752	20050000	IVAN	2	37EC8201	131D9009
1501169773	60010000	IVAN	2	3	SafeMODULE ID
1501169907	60010000	IVAN	2	3	SafeMODULE ID
1501170335	20050000	IVAN	2	7DF2A84E	131D9009
1501170810	30020000	IVAN	2	Code:Main	E916A145
1501170824	20050000	IVAN	2	7A05DFF9	C6EC4809
1501171072	60010000	IVAN	2	3	SafeMODULE ID
1501171082	20050000	IVAN	2	851B79DB	C6EC4809
1501172083	30020000	IVAN	2	Code:Main	E40FE6E7
1501172109	30010000	IVAN	2	Variables:Main	4C35EB1F
1501172121	20050000	IVAN	2	95521080	7CDCEE7F
1501172509	30020000	IVAN	2	Code:Main	5750CC40
1501172560	20050000	IVAN	2	95521080	7CDCEE7F
1501230014	30010000	IVAN	2	Variables:Main	E2AC1BCE
1501230038	30020000	IVAN	2	Code:Main	E18ADEF3
1501230049	20050000	IVAN	2	851B79DB	C6EC4809
1501230333	60010000	IVAN	2	2	SafeMODULE ID
1501230352	60010000	IVAN	2	3	SafeMODULE ID
1501230359	60010000	IVAN	2	4	SafeMODULE ID
1501230376	20050000	IVAN	2	52846CC3	C6EC4809
1501233013	20050000	IVAN	2	52846CC3	C6EC4809
1501235050	60030000	IVAN	3	2	X20SI2100	SafeMODULE ID
1501235073	20050000	IVAN	2	9222EDD6	C6EC4809
1501749251	30010000	juancaf	2	Variables:Main	F69647D2
1501749257	30010000	juancaf	2	Variables:Main	3BEFD5B2
1501749366	30010000	juancaf	2	Variables:Main	382D0076
1501749396	20040000	juancaf	1	9FE6D3E0
1501749511	20040000	juancaf	1	AAA0AAA4
1501749579	30020000	juancaf	2	Code:Main	7AF19980
1501749592	30010000	juancaf	2	Variables:Main	9AAF8BCF
1501749599	30010000	juancaf	2	Variables:Main	50663ABC
1501749697	20040000	juancaf	1	E96660E3
1501749722	20040000	juancaf	1	D3715F15
1501749749	20040000	juancaf	1	E7CF2973
1501749762	20040000	juancaf	1	BC95B311
1501749804	20040000	juancaf	1	6903E131
1501749823	20040000	juancaf	1	B4ACF23C
1501749835	20040000	juancaf	1	8F7C4478
1501749861	30010000	juancaf	2	Variables:Main	D893B074
1501749864	30020000	juancaf	2	Code:Main	7F8FD50E
1501749877	20050000	juancaf	2	7DCBEFAC	47D79DCA
1501750160	30010000	juancaf	2	Variables:Main	55A25783
1501750164	30020000	juancaf	2	Code:Main	8D7B1269
1501750265	30010000	juancaf	2	Variables:Main	F1A30CD0
1501750309	30020000	juancaf	2	Code:Main	56AB40B9
1501750325	20050000	juancaf	2	4466FEB8	AE63FDAC
1501750345	30010000	juancaf	2	Variables:Main	BC2E87B5
1501750386	20040000	juancaf	1	D4843669
1501750406	30020000	juancaf	2	Code:Main	B0D0B1CF
1501750511	20040000	juancaf	1	6C15E189
1501750614	30020000	juancaf	2	Code:Main	8E4E6B45
1501750624	30010000	juancaf	2	Variables:Main	9412492D
1501750639	30020000	juancaf	2	Code:Main	68680B99
1501750729	30020000	juancaf	2	Code:Main	C028C13F
1501750910	30020000	juancaf	2	Code:Main	E73EFE22
1501752741	30020000	juancaf	2	Code:Main	890F13AF
1501752830	30020000	juancaf	2	Code:Main	E985BCD8
1501752845	20050000	juancaf	2	F111CE5A	D6FF3F11
1501752882	30010000	juancaf	2	Variables:Main	AFD5311C
1501752890	30010000	juancaf	2	Variables:Main	5C7778AC
1501753018	20040000	juancaf	1	3E31FDCF
1501753069	20040000	juancaf	1	1E8E4AA7
1501753075	30020000	juancaf	2	Code:Main	0917BAE4
1501753526	30020000	juancaf	2	Code:Main	462B4765
1501753566	30020000	juancaf	2	Code:Main	3B955A9B
1501753592	20040000	juancaf	1	0DA53AB8
1501753723	30010000	juancaf	2	Variables:Main	2054DF17
1501753751	30020000	juancaf	2	Code:Main	77876EC7
1501753761	30010000	juancaf	2	Variables:Main	D8D38723
1501753767	30020000	juancaf	2	Code:Main	3CFA4242
1501753786	20050000	juancaf	2	FD58AE65	60FF61E8
1501753845	30010000	juancaf	2	Variables:Main	1B5FCC8C
1501753902	20040000	juancaf	1	7FE5E72C
1501754077	30020000	juancaf	2	Code:Main	6B0CE35A
1501754166	30020000	juancaf	2	Code:Main	C49DEF34
1501754285	30020000	juancaf	2	Code:Main	6848FB9C
1501754322	30020000	juancaf	2	Code:Main	E379E97B
1501754353	60010000	juancaf	2	5	SafeMODULE ID
1501754420	30020000	juancaf	2	Code:Main	5F781830
1501754432	20050000	juancaf	2	1FE19EC4	327E4537
1501755002	60010000	juancaf	2	5	SafeMODULE ID
1501755017	20050000	juancaf	2	AEB48B3E	327E4537
1501756759	60010000	juancaf	2	6	SafeMODULE ID
1501756775	20050000	juancaf	2	F9F2FE3B	327E4537
1501757719	20040000	juancaf	1	4AA19C3F
1501757740	20040000	juancaf	1	9514757C
1501757794	20040000	juancaf	1	24BBBFE7
1501757812	20040000	juancaf	1	31067564
1501757837	30020000	juancaf	2	Code:Main	9969D1EE
1501757902	30010000	juancaf	2	Variables:Main	5871A052
1501757919	30010000	juancaf	2	Variables:Main	255CF04F
1501757973	30020000	juancaf	2	Code:Main	7BF82081
1501758019	30020000	juancaf	2	Code:Main	FAAF976F
1501758121	30020000	juancaf	2	Code:Main	468C011A
1501758220	30020000	juancaf	2	Code:Main	D14FF0C6
1501758245	20050000	juancaf	2	C1D530BC	8E593B5A
1501763903	30020000	juancaf	2	Code:Main	6A257F8E
1501763921	20040000	juancaf	1	DDC3E87F
1501763953	30020000	juancaf	2	Code:Main	F7B67CCC
1501763965	20050000	juancaf	2	A2D391AE	6CF35643
1501764093	20040000	juancaf	1	3A509F62
1501764152	30020000	juancaf	2	Code:Main	FE3A3140
1501764412	30020000	juancaf	2	Code:Main	2CD1FA00
1501764570	60010000	juancaf	2	1	SafeMODULE ID
1501764576	20040000	juancaf	1	93A6EA37
1501764680	20040000	juancaf	1	E543D30A
1501764695	30020000	juancaf	2	Code:Main	00868F13
1501764711	20050000	juancaf	2	8A8BB607	D4167C2F
1501768322	60010000	juancaf	2	5	SafeMODULE ID
1501768330	60010000	juancaf	2	6	SafeMODULE ID
1501768347	20050000	juancaf	2	E0C39F79	D4167C2F
1501852476	30020000	juancaf	2	Code:Main	2CAE4442
1501852510	30020000	juancaf	2	Code:Main	D0B1FEFE
1501852635	30020000	juancaf	2	Code:Main	6655F49D
1501852650	30020000	juancaf	2	Code:Main	C11AE503
1501852673	20050000	juancaf	2	572768D6	C912942B
1501853393	20050000	juancaf	2	572768D6	C912942B
1502312764	20040000	juancaf	1	4698FEA1
1502312778	30020000	juancaf	2	Code:Main	128B2A7B
1502312787	20040000	juancaf	1	A3FD93DC
1502312812	30020000	juancaf	2	Code:Main	DD695767
1502312859	20040000	juancaf	1	F2EBEDF4
1502312870	20040000	juancaf	1	D4C60EBE
1502312883	30020000	juancaf	2	Code:Main	53279999
1502313969	20050000	juancaf	2	EC0D5C26	CD45FB58
1502348784	30020000	juancaf	2	Code:Main	3F331AD4
1502348826	30020000	juancaf	2	Code:Main	1B1F1272
1502349345	30020000	juancaf	2	Code:Main	EADD9F34
1502349727	20040000	juancaf	1	A525F3A1
1502349740	20040000	juancaf	1	8E3A02B6
1502349773	30020000	juancaf	2	Code:Main	0705F2FC
1502349791	20050000	juancaf	2	92F5E1D4	ED6F6F04
1502349894	20050000	juancaf	2	92F5E1D4	ED6F6F04
1502356990	30020000	juancaf	2	Code:Main	EBBF6722
1502357153	30020000	juancaf	2	Code:Main	DDC02464
1502357307	30020000	juancaf	2	Code:Main	0D5F460F
1502357526	20040000	juancaf	1	5961695F
1502357632	30020000	juancaf	2	Code:Main	584829F7
1502357637	20040000	juancaf	1	98A52984
1502357649	20050000	juancaf	2	D6153870	1622F8A1
1502364674	20050000	juancaf	2	D6153870	1622F8A1
1502711790	30020000	IVAN	2	Code:Main	3359BDC0
1502711804	20050000	IVAN	2	5E93383E	5525C2F9
1502711876	30020000	IVAN	2	Code:Main	6EBB4D8D
1502711889	20050000	IVAN	2	E5A4DBD2	583CD154
1502712109	20040000	IVAN	1	3A509F62
1502712126	20050000	IVAN	2	594A1D70	75C07875
1502712286	20050000	IVAN	2	594A1D70	75C07875
1502713220	30020000	IVAN	2	Code:Main	04F2AD29
1502713262	20050000	IVAN	2	594A1D70	75C07875
1503051956	60010000	juancaf	2	5	SafeMODULE ID
1503051986	20050000	juancaf	2	93859501	75C07875
1503053745	60010000	juancaf	2	3	SafeMODULE ID
1503053757	20050000	juancaf	2	5CCA390D	75C07875
1504024348	20040000	juancaf	1	ACBC5551
1504024373	30020000	juancaf	2	Code:Main	93012F8D
1504024387	20050000	juancaf	2	52CBC105	1433D1BF
1504101054	20050000	juancaf	2	52CBC105	1433D1BF
1504101678	20050000	juancaf	2	52CBC105	1433D1BF
1504102790	20050000	juancaf	2	52CBC105	1433D1BF
1504794055	20050000	juancaf	2	52CBC105	1433D1BF
1504794239	30010000	juancaf	2	Variables:Main	EFB6151E
1504794393	20040000	juancaf	1	DA84ED58
1504794406	20050000	juancaf	2	C2745761	B6F5E751
1504794425	30010000	juancaf	2	Variables:Main	25EBEE7C
1504794437	30020000	juancaf	2	Code:Main	C9D365F9
1504794468	30020000	juancaf	2	Code:Main	6ABAD332
1504794469	20040000	juancaf	1	D3862D02
1504794481	20050000	juancaf	2	C64AA501	D9938FF9
1504794543	30010000	juancaf	2	Variables:Main	4672A35C
1504794574	30010000	juancaf	2	Variables:Main	B3464051
1504794592	30010000	juancaf	2	Variables:Main	A0F5E208
1504794609	30010000	juancaf	2	Variables:Main	55AD1DA7
1504794623	30010000	juancaf	2	Variables:Main	C5B61AB2
1504794635	30010000	juancaf	2	Variables:Main	B913F52A
1504794638	30020000	juancaf	2	Code:Main	9F858A8A
1504794639	20040000	juancaf	1	C3424ED6
1504794678	20040000	juancaf	1	CAD2123B
1504794714	20040000	juancaf	1	43304100
1504794726	20050000	juancaf	2	190F734D	29A38D75
1522244744	60010000	juancaf	2	1	SafeMODULE ID
1522244745	60040000	juancaf	4	X20SLX402	X20SLX402	1 - UPDATE	SafeMODULE ID
1522244997	60010000	juancaf	2	1	SafeMODULE ID
1522245017	20050000	juancaf	2	C18D2F3B	29A38D75
1522247227	20050000	juancaf	2	80BF16B7	B13A8DBE
1553089651	20050000	jorgemur	2	80BF16B7	B13A8DBE
1553785817	60010000	jorgemur	2	3	SafeMODULE ID
1553785818	60010000	jorgemur	2	4	SafeMODULE ID
1553785819	60010000	jorgemur	2	5	SafeMODULE ID
1553785820	60010000	jorgemur	2	6	SafeMODULE ID
1553785821	60010000	jorgemur	2	1	SafeMODULE ID
1553785822	60010000	jorgemur	2	2	SafeMODULE ID
1553785823	60040000	jorgemur	4	X20SI8110	X20SI8110	3 - UPDATE	SafeMODULE ID
1553785824	60040000	jorgemur	4	X20SO2110	X20SO2110	4 - UPDATE	SafeMODULE ID
1553785825	60040000	jorgemur	4	X20SI8110	X20SI8110	5 - UPDATE	SafeMODULE ID
1553785826	60040000	jorgemur	4	X20SO2110	X20SO2110	6 - UPDATE	SafeMODULE ID
1553785827	60040000	jorgemur	4	X20SLX402	X20SL8100	1	SafeMODULE ID
1553785828	60020000	jorgemur	3	2	X20SC0402	SafeMODULE ID
1553785852	60010000	jorgemur	2	1	SafeMODULE ID
1553785862	60010000	jorgemur	2	2	SafeMODULE ID
1553785875	60010000	jorgemur	2	4	SafeMODULE ID
1553785885	60010000	jorgemur	2	6	SafeMODULE ID
1553786127	20040000	jorgemur	1	21EC23C8
1553786220	20040000	jorgemur	1	9062C7D4
1553786317	20040000	jorgemur	1	170E4133
1554371274	70010100	jorgemur	1	-if tcpip -ip 192.168.127.10 -p 50000
1554372264	20050000	jorgemur	2	8601C306	0EC17010
```

### GlobalCrossReferences.csv - X20CP1382/EFI/GlobalCrossReferences.csv
```
ErrorCodeArea1,POE\Main\Code.GB,11,OUT,307,71,Write,,INT,NSQW2,,VAR_GLOBAL,GLOBAL,,
ErrorCodeArea2,POE\Main\Code.GB,26,OUT,800,82,Write,,INT,NSQW4,,VAR_GLOBAL,GLOBAL,,
Front01EStopBK1,POE\Main\Code.GB,1,IN,310,8,Read,,SAFEBOOL,SIX62.2,,VAR_GLOBAL,GLOBAL,,
Front01EStopBK2,POE\Main\Code.GB,16,IN,392,8,Read,,SAFEBOOL,SIX66.2,,VAR_GLOBAL,GLOBAL,,
Front02EStopBK1,POE\Main\Code.GB,1,IN,311,8,Read,,SAFEBOOL,SIX62.3,,VAR_GLOBAL,GLOBAL,,
Front02EStopBK2,POE\Main\Code.GB,16,IN,393,8,Read,,SAFEBOOL,SIX66.3,,VAR_GLOBAL,GLOBAL,,
g_xInputSelectMachine,POE\Main\Code.GB,16,OUT,855,37,Write,,BOOL,NSQX0.0,,VAR_GLOBAL,GLOBAL,,
GuardSwitchBK1,POE\Main\Code.GB,4,IN,312,23,Read,,SAFEBOOL,SIX62.5,,VAR_GLOBAL,GLOBAL,,
GuardSwitchBK2,POE\Main\Code.GB,19,IN,477,47,Read,,SAFEBOOL,SIX66.5,,VAR_GLOBAL,GLOBAL,,
IclaBK1Enable,POE\Main\Code.GB,29,OUT,769,81,Write,,SAFEBOOL,SQX14.1,,VAR_GLOBAL,GLOBAL,,
IclaBK2Enable,POE\Main\Code.GB,32,OUT,683,77,Write,,SAFEBOOL,SQX15.1,,VAR_GLOBAL,GLOBAL,,
InputReset,POE\Main\Code.GB,1,IN,37,83,Read,,SAFEBOOL,SIX20.0,,VAR_GLOBAL,GLOBAL,,
InputReset,POE\Main\Code.GB,2,IN,27,0,Read,,SAFEBOOL,SIX20.0,,VAR_GLOBAL,GLOBAL,,
InputReset,POE\Main\Code.GB,7,IN,155,47,Read,,SAFEBOOL,SIX20.0,,VAR_GLOBAL,GLOBAL,,
InputReset,POE\Main\Code.GB,8,IN,211,0,Read,,SAFEBOOL,SIX20.0,,VAR_GLOBAL,GLOBAL,,
InputReset,POE\Main\Code.GB,17,IN,362,30,Read,,SAFEBOOL,SIX20.0,,VAR_GLOBAL,GLOBAL,,
InputReset,POE\Main\Code.GB,20,IN,390,0,Read,,SAFEBOOL,SIX20.0,,VAR_GLOBAL,GLOBAL,,
InputReset,POE\Main\Code.GB,22,IN,547,81,Read,,SAFEBOOL,SIX20.0,,VAR_GLOBAL,GLOBAL,,
InputReset,POE\Main\Code.GB,22,IN,475,58,Read,,SAFEBOOL,SIX20.0,,VAR_GLOBAL,GLOBAL,,
InputReset,POE\Main\Code.GB,29,IN,774,15,Read,,SAFEBOOL,SIX20.0,,VAR_GLOBAL,GLOBAL,,
InputReset,POE\Main\Code.GB,29,IN,718,6,Read,,SAFEBOOL,SIX20.0,,VAR_GLOBAL,GLOBAL,,
InputReset,POE\Main\Code.GB,32,IN,652,23,Read,,SAFEBOOL,SIX20.0,,VAR_GLOBAL,GLOBAL,,
LightCurtain01BK1,POE\Main\Code.GB,7,IN,317,10,Read,,SAFEBOOL,SIX62.4,,VAR_GLOBAL,GLOBAL,,
LightCurtain01BK2,POE\Main\Code.GB,22,IN,549,3,Read,,SAFEBOOL,SIX66.4,,VAR_GLOBAL,GLOBAL,,
LightCurtain02BK1,POE\Main\Code.GB,7,IN,318,9,Read,,SAFEBOOL,SIX62.6,,VAR_GLOBAL,GLOBAL,,
LightCurtain02BK2,POE\Main\Code.GB,22,IN,559,3,Read,,SAFEBOOL,SIX66.6,,VAR_GLOBAL,GLOBAL,,
Rear01EStopBK1,POE\Main\Code.GB,1,IN,308,13,Read,,SAFEBOOL,SIX62.0,,VAR_GLOBAL,GLOBAL,,
Rear01EStopBK2,POE\Main\Code.GB,16,IN,394,49,Read,,SAFEBOOL,SIX66.0,,VAR_GLOBAL,GLOBAL,,
Rear02EStopBK1,POE\Main\Code.GB,1,IN,309,13,Read,,SAFEBOOL,SIX62.1,,VAR_GLOBAL,GLOBAL,,
Rear02EStopBK2,POE\Main\Code.GB,16,IN,395,49,Read,,SAFEBOOL,SIX66.1,,VAR_GLOBAL,GLOBAL,,
ReleaseIclaBK1,POE\Main\Code.GB,30,OUT,773,78,Write,,BOOL,NSQX133.1,,VAR_GLOBAL,GLOBAL,,
ReleaseIclaBK2,POE\Main\Code.GB,33,OUT,689,81,Write,,BOOL,NSQX134.1,,VAR_GLOBAL,GLOBAL,,
ReleaseTransport,POE\Main\Code.GB,27,OUT,719,66,Write,,BOOL,NSQX132.0,,VAR_GLOBAL,GLOBAL,,
ReleaseUpDownBK1,POE\Main\Code.GB,30,OUT,772,74,Write,,BOOL,NSQX133.0,,VAR_GLOBAL,GLOBAL,,
ReleaseUpDownBK2,POE\Main\Code.GB,33,OUT,688,77,Write,,BOOL,NSQX134.0,,VAR_GLOBAL,GLOBAL,,
SelectMachine,POE\Main\Code.GB,16,IN,801,53,Read,,SAFEBOOL,SIX69.0,,VAR_GLOBAL,GLOBAL,,
SelectMachine,POE\Main\Code.GB,16,IN,804,12,Read,,SAFEBOOL,SIX69.0,,VAR_GLOBAL,GLOBAL,,
SelectMachine,POE\Main\Code.GB,16,IN,856,10,Read,,SAFEBOOL,SIX69.0,,VAR_GLOBAL,GLOBAL,,
SelectMachine,POE\Main\Code.GB,17,IN,802,29,Read,,SAFEBOOL,SIX69.0,,VAR_GLOBAL,GLOBAL,,
SelectMachine,POE\Main\Code.GB,17,IN,803,0,Read,,SAFEBOOL,SIX69.0,,VAR_GLOBAL,GLOBAL,,
SelectMachine,POE\Main\Code.GB,19,IN,805,57,Read,,SAFEBOOL,SIX69.0,,VAR_GLOBAL,GLOBAL,,
SelectMachine,POE\Main\Code.GB,22,IN,806,8,Read,,SAFEBOOL,SIX69.0,,VAR_GLOBAL,GLOBAL,,
SelectMachine,POE\Main\Code.GB,22,IN,807,80,Read,,SAFEBOOL,SIX69.0,,VAR_GLOBAL,GLOBAL,,
SelectMachine,POE\Main\Code.GB,25,IN,812,23,Read,,SAFEBOOL,SIX69.0,,VAR_GLOBAL,GLOBAL,,
SelectMachine,POE\Main\Code.GB,28,IN,835,5,Read,,SAFEBOOL,SIX69.0,,VAR_GLOBAL,GLOBAL,,
TransportEnable,POE\Main\Code.GB,25,OUT,716,0,Write,,SAFEBOOL,SQX16.0,,VAR_GLOBAL,GLOBAL,,
TransportEnable,POE\Main\Code.GB,28,IN,770,44,Read,,SAFEBOOL,SQX16.0,,VAR_GLOBAL,GLOBAL,,
TransportEnable,POE\Main\Code.GB,28,IN,649,64,Read,,SAFEBOOL,SQX16.0,,VAR_GLOBAL,GLOBAL,,
UpDownBK1Enable,POE\Main\Code.GB,29,OUT,768,78,Write,,SAFEBOOL,SQX14.0,,VAR_GLOBAL,GLOBAL,,
UpDownBK2Enable,POE\Main\Code.GB,29,OUT,682,74,Write,,SAFEBOOL,SQX15.0,,VAR_GLOBAL,GLOBAL,,
```

- Safety project (password-protected, skipped)

### NODES.LST - X20CP1382/EFI/NODES.LST
```
CONFIGURATION	2	PLC		SafePCOS_31
RESOURCE	3	CPU			arm
TASKDIR	4	Tasks		SafePCOS_31	arm
TASK	5	TASK		SafePCOS_31	arm
PROGRAM	6	Main	Main	SafePCOS_31	arm
VAR_GLOBALS	4	Global_Variables	C\PLC\R\CPU\Global_Variables.VBB
VAR_GLOBALS	4	Exchange_Variables	C\PLC\R\CPU\Exchange_Variables.VBB
IO/CONFIGURATION	4	IO_Configuration	C\PLC\R\CPU\IOCONFIG.CNF
```

### RES.LST - X20CP1382/EFI/RES.LST
```
(*
NC: 1
NR: 1
NTC: 1
NTR: 1
*)
PROC	CONFIGURATION	PLC	SafePCOS_31	1
C\PLC
PROC	RESOURCE	CPU	arm
C\PLC\R\CPU
PROC	VAR_GLOBAL	Global_Variables
C\PLC\R\CPU\Global_Variables.VBB
PROC	VAR_GLOBAL	Exchange_Variables
C\PLC\R\CPU\Exchange_Variables.VBB
```
